C05441=1094.407,-79.945,449.901,175.167,15.277,152.247
C05442=1094.413,-79.695,449.891,175.169,15.278,152.247
C05443=1094.419,-79.446,449.880,175.170,15.279,152.247
C05444=1094.425,-79.197,449.869,175.172,15.279,152.247
C05445=1094.431,-78.946,449.859,175.174,15.280,152.246
C05446=1094.437,-78.696,449.848,175.175,15.280,152.246
C05447=1094.443,-78.447,449.837,175.177,15.281,152.246
C05448=1094.448,-78.197,449.826,175.179,15.282,152.246
C05449=1094.455,-77.947,449.815,175.181,15.283,152.246
C05450=1094.461,-77.698,449.805,175.182,15.284,152.245
C05451=1094.467,-77.449,449.794,175.183,15.284,152.245
C05452=1094.473,-77.199,449.783,175.185,15.285,152.245
C05453=1094.479,-76.948,449.772,175.187,15.286,152.245
C05454=1094.484,-76.699,449.762,175.189,15.286,152.244
C05455=1094.490,-76.449,449.751,175.191,15.287,152.244
C05456=1094.497,-76.200,449.740,175.192,15.288,152.244
C05457=1094.503,-75.950,449.729,175.194,15.288,152.244
C05458=1094.509,-75.700,449.718,175.195,15.289,152.244
C05459=1094.515,-75.451,449.707,175.197,15.290,152.243
C05460=1094.521,-75.201,449.696,175.199,15.291,152.243
C05461=1094.527,-74.951,449.685,175.201,15.291,152.243
C05462=1094.532,-74.702,449.674,175.203,15.292,152.243
C05463=1094.539,-74.453,449.664,175.204,15.292,152.242
C05464=1094.545,-74.202,449.653,175.205,15.293,152.242
C05465=1094.551,-73.953,449.642,175.207,15.294,152.242
C05466=1094.557,-73.703,449.631,175.209,15.295,152.242
C05467=1094.562,-73.453,449.621,175.211,15.296,152.242
C05468=1094.568,-73.203,449.610,175.213,15.297,152.241
C05469=1094.574,-72.954,449.599,175.214,15.297,152.241
C05470=1094.580,-72.704,449.588,175.215,15.298,152.241
C05471=1094.586,-72.455,449.577,175.217,15.299,152.241
C05472=1094.592,-72.204,449.566,175.219,15.299,152.241
C05473=1094.597,-71.955,449.554,175.221,15.301,152.241
C05474=1094.603,-71.705,449.543,175.223,15.301,152.240
C05475=1094.608,-71.456,449.533,175.224,15.302,152.240
C05476=1094.615,-71.205,449.521,175.225,15.302,152.240
C05477=1094.621,-70.956,449.510,175.227,15.303,152.240
C05478=1094.627,-70.707,449.499,175.229,15.304,152.239
C05479=1094.633,-70.457,449.488,175.231,15.305,152.239
C05480=1094.639,-70.207,449.477,175.233,15.306,152.239
C05481=1094.644,-69.958,449.466,175.234,15.306,152.239
C05482=1094.650,-69.708,449.455,175.236,15.308,152.239
C05483=1094.656,-69.458,449.444,175.237,15.308,152.238
C05484=1094.662,-69.209,449.433,175.239,15.308,152.238
C05485=1094.668,-68.959,449.422,175.241,15.310,152.238
C05486=1094.674,-68.709,449.411,175.242,15.310,152.238
C05487=1094.680,-68.460,449.400,175.244,15.311,152.238
C05488=1094.685,-68.210,449.388,175.246,15.312,152.237
C05489=1094.691,-67.960,449.377,175.248,15.313,152.237
C05490=1094.697,-67.710,449.366,175.250,15.314,152.237
C05491=1094.703,-67.461,449.355,175.250,15.314,152.237
C05492=1094.709,-67.211,449.343,175.252,15.315,152.237
C05493=1094.715,-66.962,449.333,175.254,15.316,152.236
C05494=1094.721,-66.712,449.322,175.256,15.317,152.236
C05495=1094.727,-66.462,449.310,175.258,15.317,152.236
C05496=1094.733,-66.212,449.300,175.260,15.318,152.236
C05497=1094.739,-65.963,449.289,175.261,15.319,152.236
C05498=1094.745,-65.713,449.276,175.263,15.320,152.235
C05499=1094.750,-65.464,449.265,175.264,15.321,152.235
C05500=1094.757,-65.213,449.254,175.266,15.321,152.235
C05501=1094.763,-64.943,449.242,175.268,15.322,152.235
C05502=1094.769,-64.674,449.231,175.270,15.323,152.235
C05503=1094.776,-64.404,449.218,175.272,15.324,152.234
C05504=1094.782,-64.134,449.206,175.274,15.325,152.234
C05505=1094.788,-63.884,449.194,175.275,15.325,152.234
C05506=1094.794,-63.634,449.184,175.277,15.326,152.234
C05507=1094.801,-63.385,449.172,175.278,15.327,152.234
C05508=1094.806,-63.135,449.161,175.280,15.328,152.233
C05509=1094.811,-62.885,449.149,175.282,15.329,152.233
C05510=1094.818,-62.635,449.138,175.284,15.330,152.233
C05511=1094.824,-62.386,449.126,175.286,15.330,152.233
C05512=1094.830,-62.136,449.115,175.287,15.332,152.233
C05513=1094.836,-61.887,449.104,175.289,15.332,152.232
C05514=1094.842,-61.636,449.093,175.291,15.333,152.232
C05515=1094.847,-61.387,449.081,175.292,15.334,152.232
C05516=1094.853,-61.138,449.070,175.294,15.334,152.232
C05517=1094.860,-60.888,449.059,175.295,15.335,152.232
C05518=1094.866,-60.639,449.047,175.297,15.336,152.231
C05519=1094.872,-60.389,449.036,175.299,15.337,152.231
C05520=1094.878,-60.139,449.025,175.301,15.338,152.231
C05521=1094.884,-59.889,449.012,175.303,15.339,152.231
C05522=1094.889,-59.640,449.002,175.304,15.339,152.230
C05523=1094.896,-59.390,448.990,175.306,15.341,152.230
C05524=1094.902,-59.141,448.979,175.308,15.341,152.230
C05525=1094.908,-58.890,448.968,175.310,15.342,152.230
C05526=1094.913,-58.641,448.956,175.311,15.343,152.230
C05527=1094.919,-58.392,448.944,175.312,15.343,152.229
C05528=1094.925,-58.142,448.933,175.314,15.344,152.229
C05529=1094.931,-57.892,448.922,175.316,15.345,152.229
C05530=1094.937,-57.642,448.910,175.318,15.346,152.229
C05531=1094.943,-57.393,448.899,175.320,15.346,152.229
C05532=1094.949,-57.143,448.887,175.321,15.348,152.228
C05533=1094.955,-56.894,448.876,175.323,15.348,152.228
C05534=1094.962,-56.643,448.865,175.325,15.349,152.228
C05535=1094.967,-56.394,448.853,175.327,15.350,152.228
C05536=1094.973,-56.144,448.841,175.329,15.351,152.228
C05537=1094.980,-55.895,448.829,175.330,15.352,152.227
C05538=1094.986,-55.645,448.819,175.332,15.353,152.227
C05539=1094.991,-55.395,448.806,175.334,15.354,152.227
C05540=1094.997,-55.146,448.795,175.336,15.354,152.227
C05541=1095.004,-54.896,448.783,175.337,15.355,152.227
C05542=1095.010,-54.647,448.772,175.339,15.355,152.226
C05543=1095.015,-54.397,448.760,175.340,15.356,152.226
C05544=1095.021,-54.147,448.749,175.342,15.357,152.226
C05545=1095.028,-53.898,448.737,175.344,15.358,152.226
C05546=1095.033,-53.648,448.725,175.346,15.359,152.225
C05547=1095.040,-53.398,448.713,175.347,15.360,152.225
C05548=1095.046,-53.148,448.702,175.349,15.361,152.225
C05549=1095.052,-52.899,448.691,175.351,15.361,152.225
C05550=1095.058,-52.649,448.679,175.353,15.363,152.225
C05551=1095.064,-52.400,448.667,175.355,15.363,152.224
C05552=1095.070,-52.150,448.656,175.356,15.364,152.224
C05553=1095.076,-51.901,448.644,175.358,15.365,152.224
C05554=1095.082,-51.650,448.633,175.360,15.366,152.224
C05555=1095.088,-51.401,448.621,175.362,15.367,152.224
C05556=1095.094,-51.151,448.610,175.363,15.368,152.223
C05557=1095.100,-50.901,448.597,175.365,15.368,152.223
C05558=1095.106,-50.652,448.586,175.367,15.370,152.223
C05559=1095.112,-50.402,448.574,175.369,15.370,152.223
C05560=1095.118,-50.153,448.562,175.371,15.371,152.223
C05561=1095.124,-49.903,448.551,175.371,15.372,152.223
C05562=1095.129,-49.654,448.539,175.373,15.372,152.222
C05563=1095.136,-49.404,448.527,175.375,15.373,152.222
C05564=1095.141,-49.154,448.515,175.377,15.374,152.222
C05565=1095.147,-48.885,448.503,175.379,15.376,152.222
C05566=1095.153,-48.616,448.489,175.381,15.377,152.222
C05567=1095.160,-48.347,448.477,175.383,15.377,152.221
C05568=1095.166,-48.080,448.464,175.385,15.378,152.221
C05569=1095.172,-47.829,448.452,175.386,15.379,152.221
C05570=1095.178,-47.580,448.441,175.388,15.380,152.221
C05571=1095.184,-47.330,448.428,175.390,15.381,152.221
C05572=1095.190,-47.080,448.417,175.392,15.382,152.220
C05573=1095.195,-46.831,448.405,175.393,15.383,152.220
C05574=1095.202,-46.581,448.393,175.395,15.384,152.220
C05575=1095.207,-46.332,448.381,175.397,15.385,152.220
C05576=1095.214,-46.082,448.369,175.399,15.386,152.220
C05577=1095.219,-45.833,448.357,175.400,15.387,152.219
C05578=1095.225,-45.583,448.345,175.402,15.387,152.219
C05579=1095.231,-45.333,448.333,175.404,15.388,152.219
C05580=1095.237,-45.084,448.321,175.406,15.389,152.219
C05581=1095.243,-44.834,448.309,175.408,15.390,152.219
C05582=1095.248,-44.584,448.298,175.409,15.391,152.218
C05583=1095.255,-44.335,448.286,175.411,15.392,152.218
C05584=1095.261,-44.085,448.273,175.413,15.393,152.218
C05585=1095.266,-43.836,448.261,175.415,15.394,152.218
C05586=1095.272,-43.585,448.250,175.416,15.394,152.218
C05587=1095.278,-43.335,448.237,175.418,15.396,152.217
C05588=1095.284,-43.087,448.226,175.420,15.396,152.217
C05589=1095.290,-42.837,448.213,175.421,15.398,152.217
C05590=1095.295,-42.587,448.202,175.423,15.398,152.217
C05591=1095.302,-42.337,448.190,175.425,15.399,152.217
C05592=1095.308,-42.087,448.177,175.427,15.400,152.216
C05593=1095.313,-41.838,448.165,175.429,15.401,152.216
C05594=1095.320,-41.589,448.153,175.430,15.402,152.216
C05595=1095.326,-41.339,448.140,175.432,15.403,152.216
C05596=1095.331,-41.089,448.129,175.434,15.404,152.216
C05597=1095.337,-40.839,448.117,175.436,15.405,152.216
C05598=1095.343,-40.590,448.104,175.438,15.405,152.215
C05599=1095.349,-40.341,448.093,175.439,15.406,152.215
C05600=1095.355,-40.091,448.080,175.441,15.407,152.215
C05601=1095.361,-39.841,448.068,175.443,15.408,152.215
C05602=1095.367,-39.591,448.057,175.445,15.409,152.215
C05603=1095.373,-39.342,448.044,175.446,15.410,152.214
C05604=1095.379,-39.092,448.032,175.448,15.411,152.214
C05605=1095.385,-38.842,448.020,175.450,15.412,152.214
C05606=1095.391,-38.593,448.008,175.451,15.413,152.214
C05607=1095.397,-38.343,447.995,175.453,15.414,152.214
C05608=1095.402,-38.094,447.983,175.455,15.415,152.213
C05609=1095.409,-37.844,447.971,175.457,15.415,152.213
C05610=1095.414,-37.594,447.958,175.458,15.417,152.213
C05611=1095.420,-37.345,447.946,175.460,15.417,152.213
C05612=1095.425,-37.095,447.934,175.462,15.418,152.213
C05613=1095.431,-36.845,447.922,175.464,15.419,152.212
C05614=1095.437,-36.596,447.910,175.466,15.420,152.212
C05615=1095.443,-36.346,447.898,175.467,15.421,152.212
C05616=1095.449,-36.096,447.885,175.469,15.422,152.212
C05617=1095.454,-35.847,447.873,175.471,15.424,152.212
C05618=1095.460,-35.597,447.860,175.473,15.424,152.211
C05619=1095.467,-35.348,447.848,175.475,15.425,152.211
C05620=1095.473,-35.098,447.836,175.477,15.426,152.211
C05621=1095.478,-34.848,447.824,175.478,15.427,152.211
C05622=1095.484,-34.599,447.811,175.480,15.428,152.211
C05623=1095.490,-34.349,447.798,175.482,15.429,152.211
C05624=1095.495,-34.100,447.786,175.484,15.430,152.210
C05625=1095.501,-33.850,447.774,175.486,15.431,152.210
C05626=1095.508,-33.600,447.762,175.487,15.432,152.210
C05627=1095.514,-33.350,447.749,175.489,15.433,152.210
C05628=1095.519,-33.101,447.737,175.491,15.434,152.210
C05629=1095.526,-32.832,447.724,175.493,15.434,152.209
C05630=1095.532,-32.564,447.710,175.494,15.436,152.209
C05631=1095.538,-32.296,447.696,175.497,15.437,152.209
C05632=1095.545,-32.028,447.683,175.499,15.438,152.209
C05633=1095.550,-31.769,447.670,175.500,15.439,152.209
C05634=1095.557,-31.512,447.658,175.502,15.439,152.208
C05635=1095.563,-31.253,447.645,175.504,15.441,152.208
C05636=1095.569,-30.996,447.631,175.506,15.441,152.208
C05637=1095.575,-30.746,447.619,175.507,15.443,152.208
C05638=1095.581,-30.497,447.607,175.510,15.444,152.208
C05639=1095.587,-30.247,447.594,175.512,15.445,152.207
C05640=1095.593,-29.997,447.582,175.513,15.446,152.207
C05641=1095.598,-29.747,447.569,175.515,15.446,152.207
C05642=1095.604,-29.498,447.557,175.517,15.448,152.207
C05643=1095.610,-29.249,447.544,175.519,15.448,152.207
C05644=1095.616,-28.999,447.531,175.521,15.449,152.206
C05645=1095.622,-28.749,447.519,175.522,15.450,152.206
C05646=1095.628,-28.499,447.506,175.524,15.451,152.206
C05647=1095.633,-28.250,447.494,175.526,15.452,152.206
C05648=1095.640,-28.001,447.481,175.528,15.453,152.206
C05649=1095.646,-27.751,447.469,175.529,15.454,152.206
C05650=1095.652,-27.501,447.456,175.531,15.455,152.205
C05651=1095.658,-27.251,447.444,175.533,15.455,152.205
C05652=1095.664,-27.002,447.431,175.535,15.457,152.205
C05653=1095.669,-26.753,447.418,175.537,15.458,152.205
C05654=1095.675,-26.503,447.406,175.539,15.459,152.205
C05655=1095.681,-26.253,447.393,175.541,15.460,152.204
C05656=1095.686,-26.003,447.380,175.542,15.461,152.204
C05657=1095.692,-25.754,447.367,175.544,15.462,152.204
C05658=1095.698,-25.505,447.354,175.546,15.463,152.204
C05659=1095.704,-25.255,447.342,175.548,15.464,152.204
C05660=1095.709,-25.005,447.329,175.550,15.464,152.203
C05661=1095.716,-24.756,447.316,175.551,15.465,152.203
C05662=1095.722,-24.506,447.304,175.553,15.466,152.203
C05663=1095.727,-24.256,447.291,175.555,15.468,152.203
C05664=1095.733,-24.007,447.279,175.557,15.469,152.203
C05665=1095.739,-23.757,447.266,175.559,15.470,152.202
C05666=1095.744,-23.507,447.252,175.561,15.471,152.202
C05667=1095.750,-23.257,447.240,175.562,15.472,152.202
C05668=1095.756,-23.008,447.227,175.564,15.472,152.202
C05669=1095.762,-22.759,447.214,175.566,15.474,152.202
C05670=1095.768,-22.509,447.202,175.568,15.474,152.201
C05671=1095.774,-22.260,447.189,175.570,15.475,152.201
C05672=1095.780,-22.010,447.176,175.572,15.477,152.201
C05673=1095.786,-21.760,447.163,175.574,15.477,152.201
C05674=1095.791,-21.510,447.150,175.575,15.479,152.201
C05675=1095.796,-21.261,447.137,175.577,15.479,152.200
C05676=1095.803,-21.012,447.124,175.579,15.481,152.200
C05677=1095.808,-20.762,447.112,175.581,15.481,152.200
C05678=1095.814,-20.512,447.099,175.583,15.482,152.200
C05679=1095.821,-20.263,447.086,175.584,15.483,152.200
C05680=1095.826,-20.013,447.073,175.586,15.484,152.200
C05681=1095.832,-19.763,447.059,175.588,15.486,152.199
C05682=1095.838,-19.514,447.047,175.590,15.486,152.199
C05683=1095.844,-19.264,447.034,175.592,15.488,152.199
C05684=1095.850,-19.014,447.021,175.594,15.488,152.199
C05685=1095.855,-18.765,447.009,175.596,15.489,152.199
C05686=1095.861,-18.516,446.995,175.597,15.490,152.198
C05687=1095.867,-18.266,446.982,175.599,15.491,152.198
C05688=1095.873,-18.016,446.969,175.601,15.492,152.198
C05689=1095.879,-17.767,446.957,175.603,15.493,152.198
C05690=1095.885,-17.517,446.943,175.605,15.494,152.197
C05691=1095.890,-17.267,446.930,175.607,15.495,152.197
C05692=1095.896,-17.018,446.917,175.609,15.496,152.197
C05693=1095.902,-16.757,446.903,175.610,15.497,152.197
C05694=1095.909,-16.496,446.889,175.612,15.498,152.197
C05695=1095.915,-16.235,446.876,175.614,15.499,152.197
C05696=1095.921,-15.975,446.862,175.617,15.500,152.196
C05697=1095.927,-15.725,446.850,175.618,15.501,152.196
C05698=1095.933,-15.476,446.836,175.620,15.502,152.196
C05699=1095.939,-15.226,446.824,175.622,15.503,152.196
C05700=1095.944,-14.976,446.810,175.624,15.504,152.196
C05701=1095.950,-14.726,446.797,175.625,15.505,152.195
C05702=1095.956,-14.477,446.784,175.628,15.506,152.195
C05703=1095.961,-14.227,446.771,175.630,15.507,152.195
C05704=1095.968,-13.977,446.758,175.631,15.508,152.195
C05705=1095.974,-13.728,446.744,175.633,15.509,152.195
C05706=1095.979,-13.478,446.731,175.635,15.510,152.194
C05707=1095.985,-13.229,446.718,175.637,15.511,152.194
C05708=1095.990,-12.979,446.705,175.638,15.512,152.194
C05709=1095.997,-12.729,446.692,175.641,15.513,152.194
C05710=1096.003,-12.480,446.678,175.643,15.514,152.194
C05711=1096.008,-12.230,446.665,175.645,15.515,152.193
C05712=1096.014,-11.981,446.652,175.646,15.516,152.193
C05713=1096.019,-11.732,446.638,175.648,15.517,152.193
C05714=1096.025,-11.482,446.626,175.650,15.518,152.193
C05715=1096.031,-11.233,446.613,175.652,15.519,152.193
C05716=1096.037,-10.983,446.599,175.654,15.520,152.192
C05717=1096.043,-10.733,446.586,175.656,15.521,152.192
C05718=1096.048,-10.484,446.572,175.658,15.522,152.192
C05719=1096.054,-10.234,446.559,175.660,15.523,152.192
C05720=1096.059,-9.984,446.546,175.661,15.524,152.192
C05721=1096.066,-9.735,446.533,175.663,15.525,152.191
C05722=1096.072,-9.486,446.519,175.666,15.526,152.191
C05723=1096.077,-9.236,446.505,175.667,15.527,152.191
C05724=1096.083,-8.986,446.493,175.669,15.528,152.191
C05725=1096.089,-8.737,446.479,175.671,15.528,152.191
C05726=1096.095,-8.487,446.466,175.673,15.530,152.190
C05727=1096.100,-8.238,446.452,175.675,15.530,152.190
C05728=1096.107,-7.987,446.439,175.677,15.532,152.190
C05729=1096.112,-7.738,446.425,175.679,15.533,152.190
C05730=1096.119,-7.488,446.412,175.681,15.534,152.190
C05731=1096.124,-7.239,446.398,175.682,15.535,152.189
C05732=1096.130,-6.989,446.385,175.684,15.535,152.189
C05733=1096.136,-6.739,446.372,175.686,15.536,152.189
C05734=1096.142,-6.490,446.358,175.688,15.538,152.189
C05735=1096.147,-6.240,446.344,175.690,15.539,152.189
C05736=1096.153,-5.991,446.331,175.692,15.539,152.188
C05737=1096.159,-5.742,446.317,175.694,15.541,152.188
C05738=1096.165,-5.492,446.305,175.696,15.541,152.188
C05739=1096.170,-5.242,446.291,175.698,15.542,152.188
C05740=1096.176,-4.993,446.278,175.700,15.544,152.188
C05741=1096.182,-4.743,446.264,175.702,15.544,152.187
C05742=1096.188,-4.494,446.250,175.704,15.545,152.187
C05743=1096.194,-4.244,446.236,175.705,15.546,152.187
C05744=1096.200,-3.994,446.223,175.707,15.547,152.187
C05745=1096.206,-3.745,446.209,175.709,15.548,152.186
C05746=1096.212,-3.495,446.197,175.711,15.549,152.186
C05747=1096.217,-3.245,446.183,175.713,15.550,152.186
C05748=1096.224,-2.996,446.169,175.715,15.551,152.186
C05749=1096.229,-2.747,446.156,175.717,15.552,152.186
C05750=1096.234,-2.497,446.142,175.719,15.553,152.185
C05751=1096.240,-2.247,446.128,175.721,15.555,152.185
C05752=1096.246,-1.998,446.115,175.723,15.555,152.185
C05753=1096.252,-1.749,446.101,175.725,15.556,152.185
C05754=1096.257,-1.499,446.087,175.726,15.557,152.185
C05755=1096.263,-1.250,446.074,175.728,15.558,152.184
C05756=1096.269,-1.000,446.060,175.731,15.560,152.184
C05757=1096.275,-0.729,446.045,175.732,15.560,152.184
C05758=1096.281,-0.458,446.030,175.734,15.561,152.184
C05759=1096.288,-0.188,446.015,175.737,15.563,152.184
C05760=1096.294,0.084,446.000,175.739,15.564,152.183
C05761=1096.299,0.333,445.987,175.741,15.564,152.183
C05762=1096.305,0.583,445.973,175.743,15.566,152.183
C05763=1096.312,0.833,445.959,175.745,15.567,152.183
C05764=1096.317,1.082,445.945,175.747,15.568,152.182
C05765=1096.322,1.332,445.931,175.748,15.569,152.182
C05766=1096.328,1.581,445.918,175.750,15.569,152.182
C05767=1096.333,1.831,445.904,175.753,15.571,152.182
C05768=1096.340,2.080,445.890,175.754,15.572,152.182
C05769=1096.345,2.329,445.876,175.756,15.573,152.181
C05770=1096.351,2.579,445.862,175.758,15.573,152.181
C05771=1096.357,2.829,445.848,175.760,15.574,152.181
C05772=1096.363,3.078,445.834,175.762,15.576,152.181
C05773=1096.369,3.328,445.821,175.764,15.577,152.181
C05774=1096.374,3.577,445.807,175.766,15.578,152.181
C05775=1096.380,3.827,445.793,175.768,15.578,152.180
C05776=1096.385,4.077,445.779,175.770,15.579,152.180
C05777=1096.391,4.326,445.766,175.772,15.580,152.180
C05778=1096.398,4.576,445.751,175.774,15.582,152.180
C05779=1096.403,4.825,445.737,175.776,15.582,152.179
C05780=1096.409,5.075,445.723,175.778,15.583,152.179
C05781=1096.414,5.324,445.709,175.780,15.585,152.179
C05782=1096.420,5.574,445.696,175.782,15.586,152.179
C05783=1096.426,5.824,445.682,175.784,15.586,152.178
C05784=1096.432,6.073,445.667,175.786,15.587,152.178
C05785=1096.438,6.322,445.653,175.787,15.588,152.178
C05786=1096.443,6.572,445.639,175.790,15.589,152.178
C05787=1096.449,6.821,445.626,175.792,15.590,152.178
C05788=1096.455,7.071,445.612,175.793,15.591,152.177
C05789=1096.461,7.320,445.597,175.795,15.592,152.177
C05790=1096.467,7.570,445.583,175.798,15.593,152.177
C05791=1096.472,7.820,445.570,175.800,15.594,152.177
C05792=1096.478,8.070,445.555,175.801,15.595,152.177
C05793=1096.484,8.319,445.541,175.803,15.596,152.176
C05794=1096.489,8.568,445.527,175.805,15.597,152.176
C05795=1096.496,8.818,445.514,175.808,15.598,152.176
C05796=1096.502,9.068,445.499,175.810,15.599,152.176
C05797=1096.508,9.317,445.485,175.811,15.600,152.175
C05798=1096.513,9.566,445.471,175.813,15.601,152.175
C05799=1096.519,9.816,445.457,175.816,15.602,152.175
C05800=1096.525,10.066,445.442,175.818,15.603,152.175
C05801=1096.530,10.315,445.428,175.819,15.604,152.175
C05802=1096.536,10.565,445.414,175.821,15.604,152.174
C05803=1096.542,10.814,445.400,175.824,15.606,152.174
C05804=1096.548,11.064,445.386,175.826,15.606,152.174
C05805=1096.554,11.313,445.372,175.828,15.607,152.173
C05806=1096.560,11.562,445.358,175.829,15.608,152.173
C05807=1096.566,11.813,445.344,175.832,15.610,152.173
C05808=1096.571,12.062,445.330,175.834,15.610,152.173
C05809=1096.577,12.311,445.315,175.836,15.611,152.173
C05810=1096.583,12.561,445.301,175.838,15.612,152.172
C05811=1096.589,12.810,445.286,175.840,15.613,152.172
C05812=1096.594,13.060,445.272,175.842,15.614,152.172
C05813=1096.600,13.310,445.258,175.844,15.615,152.172
C05814=1096.606,13.559,445.244,175.846,15.616,152.171
C05815=1096.612,13.809,445.230,175.848,15.616,152.171
C05816=1096.618,14.058,445.215,175.850,15.618,152.171
C05817=1096.624,14.308,445.202,175.852,15.618,152.171
C05818=1096.629,14.557,445.186,175.854,15.619,152.170
C05819=1096.635,14.807,445.172,175.856,15.620,152.170
C05820=1096.641,15.056,445.158,175.858,15.622,152.170
C05821=1096.648,15.329,445.142,175.860,15.622,152.170
C05822=1096.654,15.601,445.127,175.863,15.624,152.169
C05823=1096.660,15.874,445.111,175.865,15.624,152.169
C05824=1096.667,16.147,445.095,175.867,15.626,152.169
C05825=1096.672,16.397,445.081,175.869,15.627,152.169
C05826=1096.678,16.646,445.066,175.871,15.628,152.169
C05827=1096.684,16.896,445.052,175.873,15.628,152.168
C05828=1096.689,17.145,445.037,175.875,15.630,152.168
C05829=1096.695,17.395,445.023,175.877,15.630,152.168
C05830=1096.701,17.645,445.008,175.879,15.631,152.167
C05831=1096.706,17.894,444.994,175.881,15.632,152.167
C05832=1096.712,18.143,444.980,175.883,15.634,152.167
C05833=1096.718,18.393,444.965,175.885,15.634,152.167
C05834=1096.724,18.642,444.951,175.887,15.635,152.167
C05835=1096.730,18.891,444.936,175.890,15.636,152.166
C05836=1096.735,19.142,444.921,175.892,15.637,152.166
C05837=1096.741,19.391,444.907,175.894,15.638,152.166
C05838=1096.747,19.641,444.893,175.896,15.638,152.166
C05839=1096.753,19.890,444.878,175.898,15.640,152.165
C05840=1096.759,20.139,444.864,175.900,15.641,152.165
C05841=1096.765,20.389,444.849,175.902,15.642,152.165
C05842=1096.770,20.639,444.834,175.904,15.642,152.165
C05843=1096.776,20.888,444.820,175.906,15.644,152.164
C05844=1096.782,21.138,444.805,175.908,15.644,152.164
C05845=1096.787,21.387,444.791,175.910,15.645,152.164
C05846=1096.793,21.637,444.775,175.913,15.646,152.164
C05847=1096.799,21.886,444.761,175.914,15.648,152.163
C05848=1096.804,22.135,444.747,175.916,15.648,152.163
C05849=1096.811,22.385,444.732,175.918,15.649,152.163
C05850=1096.815,22.635,444.717,175.921,15.650,152.163
C05851=1096.822,22.885,444.702,175.923,15.651,152.162
C05852=1096.828,23.134,444.688,175.925,15.652,152.162
C05853=1096.832,23.383,444.673,175.927,15.653,152.162
C05854=1096.839,23.633,444.658,175.929,15.654,152.162
C05855=1096.844,23.882,444.644,175.931,15.654,152.161
C05856=1096.851,24.132,444.629,175.933,15.655,152.161
C05857=1096.856,24.382,444.614,175.936,15.656,152.161
C05858=1096.862,24.631,444.599,175.937,15.658,152.161
C05859=1096.868,24.880,444.585,175.939,15.658,152.161
C05860=1096.873,25.130,444.569,175.942,15.660,152.160
C05861=1096.879,25.379,444.555,175.944,15.660,152.160
C05862=1096.885,25.629,444.541,175.945,15.661,152.160
C05863=1096.890,25.879,444.525,175.947,15.662,152.159
C05864=1096.896,26.128,444.511,175.950,15.663,152.159
C05865=1096.902,26.377,444.496,175.952,15.664,152.159
C05866=1096.908,26.627,444.481,175.954,15.665,152.159
C05867=1096.914,26.876,444.466,175.956,15.666,152.158
C05868=1096.919,27.126,444.452,175.958,15.667,152.158
C05869=1096.925,27.376,444.436,175.960,15.667,152.158
C05870=1096.931,27.625,444.422,175.963,15.669,152.158
C05871=1096.937,27.874,444.407,175.965,15.669,152.157
C05872=1096.942,28.124,444.392,175.967,15.670,152.157
C05873=1096.949,28.373,444.377,175.969,15.671,152.157
C05874=1096.954,28.622,444.362,175.971,15.672,152.157
C05875=1096.960,28.872,444.347,175.973,15.673,152.156
C05876=1096.966,29.122,444.333,175.975,15.673,152.156
C05877=1096.971,29.372,444.317,175.978,15.675,152.156
C05878=1096.977,29.621,444.303,175.980,15.676,152.155
C05879=1096.983,29.871,444.287,175.981,15.676,152.155
C05880=1096.988,30.120,444.272,175.984,15.678,152.155
C05881=1096.994,30.370,444.257,175.986,15.678,152.155
C05882=1097.000,30.619,444.242,175.988,15.679,152.154
C05883=1097.005,30.868,444.227,175.991,15.680,152.154
C05884=1097.011,31.117,444.212,175.992,15.681,152.154
C05885=1097.017,31.392,444.195,175.994,15.682,152.154
C05886=1097.023,31.666,444.179,175.997,15.683,152.153
C05887=1097.030,31.940,444.162,176.000,15.684,152.153
C05888=1097.037,32.214,444.146,176.002,15.685,152.153
C05889=1097.042,32.464,444.130,176.003,15.686,152.153
C05890=1097.048,32.713,444.116,176.006,15.687,152.152
C05891=1097.054,32.963,444.100,176.008,15.688,152.152
C05892=1097.059,33.212,444.085,176.010,15.688,152.152
C05893=1097.065,33.462,444.070,176.013,15.689,152.151
C05894=1097.070,33.711,444.055,176.015,15.690,152.151
C05895=1097.076,33.961,444.040,176.017,15.691,152.151
C05896=1097.082,34.211,444.025,176.019,15.692,152.151
C05897=1097.088,34.460,444.010,176.021,15.693,152.150
C05898=1097.094,34.709,443.994,176.023,15.694,152.150
C05899=1097.100,34.958,443.979,176.026,15.695,152.150
C05900=1097.105,35.208,443.964,176.028,15.696,152.150
C05901=1097.111,35.457,443.949,176.030,15.696,152.149
C05902=1097.117,35.707,443.933,176.032,15.698,152.149
C05903=1097.122,35.957,443.918,176.034,15.698,152.149
C05904=1097.128,36.206,443.903,176.036,15.699,152.148
C05905=1097.134,36.456,443.888,176.039,15.700,152.148
C05906=1097.140,36.704,443.872,176.041,15.701,152.148
C05907=1097.145,36.954,443.857,176.043,15.701,152.148
C05908=1097.151,37.204,443.841,176.045,15.703,152.147
C05909=1097.157,37.453,443.827,176.047,15.703,152.147
C05910=1097.163,37.703,443.811,176.049,15.704,152.147
C05911=1097.169,37.952,443.796,176.052,15.705,152.146
C05912=1097.174,38.201,443.780,176.054,15.706,152.146
C05913=1097.180,38.451,443.765,176.056,15.706,152.146
C05914=1097.185,38.701,443.750,176.059,15.708,152.146
C05915=1097.191,38.950,443.735,176.060,15.708,152.145
C05916=1097.197,39.200,443.719,176.062,15.709,152.145
C05917=1097.202,39.449,443.703,176.065,15.710,152.145
C05918=1097.209,39.699,443.688,176.067,15.711,152.144
C05919=1097.214,39.948,443.673,176.069,15.712,152.144
C05920=1097.220,40.197,443.657,176.072,15.713,152.144
C05921=1097.225,40.447,443.641,176.074,15.713,152.144
C05922=1097.231,40.696,443.627,176.076,15.714,152.143
C05923=1097.237,40.945,443.611,176.078,15.715,152.143
C05924=1097.243,41.195,443.595,176.080,15.716,152.143
C05925=1097.248,41.445,443.580,176.083,15.717,152.142
C05926=1097.253,41.695,443.564,176.085,15.718,152.142
C05927=1097.260,41.943,443.549,176.087,15.718,152.142
C05928=1097.265,42.193,443.533,176.090,15.720,152.142
C05929=1097.271,42.442,443.517,176.091,15.720,152.141
C05930=1097.276,42.692,443.502,176.093,15.721,152.141
C05931=1097.283,42.941,443.487,176.096,15.722,152.141
C05932=1097.288,43.191,443.471,176.098,15.723,152.140
C05933=1097.294,43.441,443.455,176.100,15.723,152.140
C05934=1097.299,43.690,443.440,176.103,15.725,152.140
C05935=1097.305,43.939,443.424,176.105,15.725,152.140
C05936=1097.311,44.189,443.408,176.107,15.726,152.139
C05937=1097.316,44.438,443.392,176.109,15.727,152.139
C05938=1097.322,44.688,443.377,176.111,15.728,152.139
C05939=1097.327,44.937,443.362,176.114,15.729,152.138
C05940=1097.334,45.186,443.346,176.116,15.730,152.138
C05941=1097.339,45.436,443.331,176.118,15.730,152.138
C05942=1097.345,45.685,443.315,176.121,15.731,152.137
C05943=1097.350,45.935,443.299,176.123,15.732,152.137
C05944=1097.356,46.184,443.283,176.125,15.733,152.137
C05945=1097.361,46.433,443.268,176.127,15.734,152.137
C05946=1097.367,46.683,443.251,176.129,15.735,152.136
C05947=1097.373,46.933,443.236,176.132,15.736,152.136
C05948=1097.378,47.181,443.220,176.134,15.736,152.136
C05949=1097.384,47.456,443.202,176.137,15.738,152.135
C05950=1097.390,47.730,443.185,176.139,15.738,152.135
C05951=1097.397,48.005,443.168,176.141,15.739,152.135
C05952=1097.403,48.279,443.150,176.143,15.740,152.134
C05953=1097.408,48.528,443.135,176.146,15.741,152.134
C05954=1097.414,48.778,443.118,176.148,15.741,152.134
C05955=1097.420,49.028,443.103,176.151,15.743,152.133
C05956=1097.426,49.277,443.087,176.153,15.743,152.133
C05957=1097.431,49.526,443.071,176.155,15.744,152.133
C05958=1097.437,49.776,443.055,176.158,15.745,152.132
C05959=1097.442,50.025,443.039,176.159,15.746,152.132
C05960=1097.448,50.275,443.023,176.162,15.746,152.132
C05961=1097.453,50.524,443.007,176.164,15.747,152.132
C05962=1097.459,50.773,442.992,176.166,15.748,152.131
C05963=1097.465,51.023,442.976,176.169,15.749,152.131
C05964=1097.471,51.272,442.959,176.171,15.750,152.131
C05965=1097.476,51.521,442.944,176.173,15.750,152.130
C05966=1097.482,51.771,442.928,176.176,15.751,152.130
C05967=1097.488,52.020,442.912,176.178,15.752,152.130
C05968=1097.494,52.270,442.896,176.181,15.753,152.129
C05969=1097.500,52.519,442.880,176.183,15.753,152.129
C05970=1097.505,52.768,442.864,176.185,15.754,152.129
C05971=1097.511,53.018,442.848,176.188,15.755,152.128
C05972=1097.517,53.267,442.832,176.189,15.756,152.128
C05973=1097.522,53.517,442.815,176.192,15.757,152.128
C05974=1097.528,53.766,442.799,176.194,15.757,152.127
C05975=1097.533,54.016,442.784,176.196,15.758,152.127
C05976=1097.539,54.265,442.768,176.199,15.759,152.127
C05977=1097.545,54.514,442.751,176.201,15.760,152.126
C05978=1097.551,54.764,442.735,176.203,15.760,152.126
C05979=1097.556,55.014,442.720,176.206,15.761,152.126
C05980=1097.562,55.263,442.703,176.208,15.762,152.125
C05981=1097.568,55.512,442.687,176.211,15.763,152.125
C05982=1097.573,55.761,442.671,176.213,15.763,152.125
C05983=1097.579,56.011,442.654,176.215,15.764,152.124
C05984=1097.584,56.261,442.639,176.218,15.765,152.124
C05985=1097.590,56.510,442.623,176.220,15.765,152.124
C05986=1097.596,56.759,442.606,176.222,15.767,152.123
C05987=1097.602,57.009,442.590,176.225,15.767,152.123
C05988=1097.608,57.258,442.574,176.226,15.768,152.123
C05989=1097.614,57.507,442.558,176.229,15.768,152.122
C05990=1097.619,57.756,442.541,176.231,15.769,152.122
C05991=1097.624,58.006,442.526,176.234,15.770,152.122
C05992=1097.630,58.256,442.509,176.236,15.771,152.121
C05993=1097.636,58.505,442.493,176.238,15.771,152.121
C05994=1097.642,58.754,442.477,176.241,15.772,152.121
C05995=1097.648,59.004,442.461,176.243,15.772,152.120
C05996=1097.653,59.253,442.444,176.246,15.774,152.120
C05997=1097.659,59.503,442.427,176.248,15.774,152.120
C05998=1097.665,59.752,442.411,176.251,15.775,152.119
C05999=1097.671,60.001,442.395,176.253,15.776,152.119
C06000=1097.677,60.251,442.379,176.255,15.776,152.118
C06001=1097.683,60.500,442.362,176.258,15.777,152.118
C06002=1097.688,60.750,442.346,176.260,15.777,152.118
C06003=1097.694,60.999,442.329,176.263,15.779,152.117
C06004=1097.700,61.249,442.313,176.265,15.779,152.117
C06005=1097.706,61.498,442.297,176.267,15.779,152.117
C06006=1097.711,61.748,442.280,176.270,15.781,152.116
C06007=1097.717,61.997,442.264,176.272,15.781,152.116
C06008=1097.723,62.246,442.247,176.275,15.782,152.116
C06009=1097.729,62.496,442.231,176.277,15.782,152.115
C06010=1097.735,62.745,442.215,176.279,15.783,152.115
C06011=1097.740,62.995,442.198,176.282,15.783,152.114
C06012=1097.746,63.244,442.182,176.284,15.784,152.114
C06013=1097.753,63.517,442.164,176.287,15.785,152.114
C06014=1097.759,63.792,442.146,176.290,15.786,152.113
C06015=1097.765,64.066,442.127,176.292,15.786,152.113
C06016=1097.772,64.340,442.109,176.295,15.787,152.112
C06017=1097.777,64.590,442.093,176.297,15.788,152.112
C06018=1097.783,64.839,442.076,176.300,15.789,152.112
C06019=1097.789,65.088,442.060,176.302,15.789,152.111
C06020=1097.794,65.338,442.043,176.305,15.790,152.111
C06021=1097.801,65.587,442.026,176.307,15.790,152.111
C06022=1097.806,65.836,442.009,176.309,15.791,152.110
C06023=1097.812,66.086,441.993,176.312,15.792,152.110
C06024=1097.818,66.335,441.977,176.314,15.792,152.110
C06025=1097.823,66.585,441.960,176.317,15.793,152.109
C06026=1097.829,66.834,441.944,176.319,15.794,152.109
C06027=1097.835,67.083,441.926,176.322,15.795,152.108
C06028=1097.840,67.332,441.910,176.324,15.795,152.108
C06029=1097.846,67.582,441.893,176.326,15.796,152.108
C06030=1097.852,67.831,441.877,176.329,15.797,152.107
C06031=1097.857,68.081,441.860,176.331,15.797,152.107
C06032=1097.863,68.330,441.843,176.334,15.798,152.107
C06033=1097.868,68.579,441.826,176.336,15.798,152.106
C06034=1097.874,68.829,441.810,176.339,15.799,152.106
C06035=1097.880,69.078,441.794,176.341,15.799,152.105
C06036=1097.886,69.327,441.776,176.344,15.801,152.105
C06037=1097.892,69.576,441.760,176.346,15.801,152.105
C06038=1097.897,69.826,441.743,176.348,15.801,152.104
C06039=1097.902,70.075,441.725,176.351,15.802,152.104
C06040=1097.908,70.325,441.709,176.353,15.803,152.104
C06041=1097.914,70.574,441.692,176.356,15.804,152.103
C06042=1097.920,70.823,441.675,176.358,15.804,152.103
C06043=1097.925,71.073,441.658,176.361,15.805,152.102
C06044=1097.931,71.322,441.642,176.363,15.806,152.102
C06045=1097.937,71.571,441.625,176.366,15.806,152.102
C06046=1097.942,71.821,441.607,176.368,15.807,152.101
C06047=1097.948,72.071,441.591,176.370,15.807,152.101
C06048=1097.954,72.320,441.574,176.373,15.808,152.101
C06049=1097.960,72.569,441.557,176.375,15.808,152.100
C06050=1097.965,72.819,441.541,176.378,15.809,152.100
C06051=1097.970,73.068,441.523,176.380,15.810,152.099
C06052=1097.976,73.317,441.507,176.383,15.810,152.099
C06053=1097.982,73.566,441.489,176.385,15.811,152.099
C06054=1097.987,73.816,441.472,176.388,15.812,152.098
C06055=1097.993,74.065,441.455,176.390,15.812,152.098
C06056=1097.999,74.315,441.438,176.393,15.813,152.097
C06057=1098.004,74.565,441.421,176.395,15.813,152.097
C06058=1098.011,74.813,441.404,176.397,15.814,152.097
C06059=1098.016,75.063,441.387,176.400,15.815,152.096
C06060=1098.021,75.312,441.370,176.402,15.815,152.096
C06061=1098.027,75.561,441.354,176.405,15.816,152.095
C06062=1098.033,75.810,441.336,176.408,15.816,152.095
C06063=1098.038,76.060,441.319,176.410,15.817,152.095
C06064=1098.045,76.309,441.302,176.413,15.817,152.094
C06065=1098.050,76.559,441.285,176.416,15.818,152.094
C06066=1098.056,76.808,441.267,176.418,15.819,152.093
C06067=1098.062,77.057,441.250,176.421,15.819,152.093
C06068=1098.067,77.307,441.234,176.423,15.820,152.093
C06069=1098.073,77.556,441.216,176.425,15.820,152.092
C06070=1098.079,77.806,441.199,176.428,15.821,152.092
C06071=1098.085,78.055,441.182,176.430,15.821,152.091
C06072=1098.090,78.304,441.165,176.433,15.822,152.091
C06073=1098.096,78.553,441.147,176.435,15.823,152.091
C06074=1098.101,78.802,441.130,176.438,15.824,152.090
C06075=1098.108,79.052,441.113,176.440,15.824,152.090
C06076=1098.113,79.302,441.096,176.443,15.825,152.089
C06077=1098.119,79.575,441.077,176.445,15.825,152.089
C06078=1098.125,79.849,441.058,176.448,15.826,152.088
C06079=1098.131,80.123,441.038,176.452,15.826,152.088
C06080=1098.137,80.397,441.020,176.455,15.827,152.087
C06081=1098.143,80.646,441.003,176.457,15.827,152.087
C06082=1098.149,80.896,440.985,176.460,15.828,152.087
C06083=1098.154,81.146,440.968,176.462,15.828,152.086
C06084=1098.160,81.395,440.950,176.465,15.829,152.086
C06085=1098.165,81.644,440.933,176.467,15.830,152.085
C06086=1098.170,81.893,440.916,176.469,15.830,152.085
C06087=1098.177,82.143,440.898,176.472,15.831,152.085
C06088=1098.183,82.392,440.881,176.475,15.831,152.084
C06089=1098.188,82.641,440.863,176.478,15.832,152.084
C06090=1098.193,82.891,440.846,176.480,15.832,152.083
C06091=1098.200,83.140,440.829,176.483,15.833,152.083
C06092=1098.205,83.389,440.811,176.485,15.833,152.082
C06093=1098.211,83.638,440.793,176.488,15.834,152.082
C06094=1098.216,83.888,440.777,176.490,15.834,152.082
C06095=1098.222,84.138,440.759,176.493,15.835,152.081
C06096=1098.227,84.387,440.741,176.495,15.835,152.081
C06097=1098.233,84.636,440.723,176.498,15.836,152.080
C06098=1098.239,84.885,440.706,176.500,15.837,152.080
C06099=1098.245,85.135,440.688,176.503,15.837,152.079
C06100=1098.250,85.384,440.671,176.505,15.838,152.079
C06101=1098.255,85.633,440.654,176.509,15.838,152.078
C06102=1098.261,85.883,440.636,176.511,15.838,152.078
C06103=1098.268,86.132,440.619,176.514,15.839,152.078
C06104=1098.273,86.381,440.601,176.516,15.839,152.077
C06105=1098.279,86.630,440.584,176.519,15.840,152.077
C06106=1098.285,86.880,440.566,176.521,15.841,152.076
C06107=1098.290,87.129,440.548,176.524,15.841,152.076
C06108=1098.296,87.378,440.530,176.527,15.841,152.075
C06109=1098.302,87.628,440.513,176.530,15.842,152.075
C06110=1098.307,87.877,440.496,176.532,15.842,152.075
C06111=1098.313,88.126,440.478,176.535,15.843,152.074
C06112=1098.319,88.376,440.460,176.537,15.843,152.074
C06113=1098.324,88.625,440.443,176.540,15.844,152.073
C06114=1098.331,88.875,440.425,176.542,15.844,152.073
C06115=1098.336,89.124,440.407,176.545,15.845,152.072
C06116=1098.341,89.373,440.389,176.548,15.845,152.072
C06117=1098.347,89.623,440.371,176.551,15.846,152.071
C06118=1098.352,89.872,440.353,176.553,15.846,152.071
C06119=1098.358,90.121,440.336,176.556,15.847,152.070
C06120=1098.364,90.371,440.318,176.558,15.847,152.070
C06121=1098.370,90.620,440.300,176.561,15.847,152.069
C06122=1098.376,90.869,440.282,176.564,15.848,152.069
C06123=1098.382,91.118,440.264,176.567,15.849,152.069
C06124=1098.387,91.367,440.247,176.569,15.849,152.068
C06125=1098.393,91.617,440.229,176.572,15.849,152.068
C06126=1098.398,91.866,440.210,176.574,15.850,152.067
C06127=1098.404,92.115,440.193,176.577,15.850,152.067
C06128=1098.410,92.365,440.175,176.579,15.851,152.066
C06129=1098.415,92.614,440.157,176.583,15.851,152.066
C06130=1098.421,92.863,440.140,176.585,15.851,152.065
C06131=1098.426,93.113,440.121,176.588,15.852,152.065
C06132=1098.432,93.362,440.104,176.590,15.852,152.065
C06133=1098.438,93.611,440.085,176.593,15.853,152.064
C06134=1098.444,93.860,440.068,176.595,15.853,152.064
C06135=1098.448,94.109,440.049,176.598,15.854,152.063
C06136=1098.454,94.359,440.031,176.601,15.854,152.063
C06137=1098.460,94.608,440.014,176.604,15.855,152.062
C06138=1098.466,94.857,439.995,176.606,15.855,152.062
C06139=1098.471,95.107,439.977,176.609,15.855,152.061
C06140=1098.477,95.356,439.960,176.612,15.856,152.061
C06141=1098.483,95.630,439.940,176.615,15.856,152.060
C06142=1098.489,95.904,439.920,176.618,15.857,152.060
C06143=1098.496,96.177,439.900,176.621,15.857,152.059
C06144=1098.502,96.451,439.880,176.623,15.858,152.059
C06145=1098.508,96.701,439.862,176.627,15.858,152.058
C06146=1098.513,96.950,439.844,176.629,15.858,152.058
C06147=1098.519,97.200,439.825,176.632,15.859,152.057
C06148=1098.524,97.449,439.808,176.634,15.859,152.057
C06149=1098.530,97.698,439.790,176.637,15.859,152.056
C06150=1098.536,97.948,439.772,176.640,15.860,152.056
C06151=1098.542,98.197,439.753,176.643,15.860,152.055
C06152=1098.547,98.446,439.735,176.645,15.860,152.055
C06153=1098.553,98.696,439.717,176.648,15.861,152.054
C06154=1098.558,98.944,439.698,176.651,15.861,152.054
C06155=1098.565,99.194,439.681,176.653,15.862,152.053
C06156=1098.570,99.443,439.662,176.656,15.862,152.053
C06157=1098.576,99.693,439.644,176.659,15.863,152.052
C06158=1098.581,99.942,439.626,176.662,15.863,152.052
C06159=1098.588,100.191,439.608,176.664,15.863,152.051
C06160=1098.592,100.440,439.589,176.668,15.864,152.051
C06161=1098.599,100.689,439.571,176.670,15.864,152.050
C06162=1098.604,100.938,439.553,176.673,15.864,152.050
C06163=1098.610,101.188,439.535,176.676,15.864,152.049
C06164=1098.616,101.438,439.516,176.679,15.865,152.049
C06165=1098.621,101.687,439.498,176.681,15.865,152.048
C06166=1098.627,101.936,439.479,176.684,15.866,152.048
C06167=1098.632,102.185,439.461,176.686,15.865,152.047
C06168=1098.639,102.434,439.442,176.689,15.866,152.047
C06169=1098.643,102.684,439.424,176.692,15.866,152.046
C06170=1098.650,102.933,439.406,176.695,15.867,152.046
C06171=1098.655,103.182,439.387,176.697,15.867,152.045
C06172=1098.661,103.431,439.369,176.700,15.868,152.045
C06173=1098.666,103.681,439.351,176.703,15.868,152.044
C06174=1098.672,103.930,439.332,176.706,15.868,152.044
C06175=1098.677,104.179,439.314,176.709,15.869,152.043
C06176=1098.683,104.428,439.295,176.711,15.869,152.043
C06177=1098.689,104.677,439.276,176.715,15.869,152.042
C06178=1098.694,104.927,439.258,176.717,15.869,152.042
C06179=1098.700,105.176,439.239,176.720,15.870,152.041
C06180=1098.705,105.426,439.221,176.722,15.870,152.041
C06181=1098.712,105.675,439.202,176.725,15.871,152.040
C06182=1098.717,105.923,439.183,176.728,15.871,152.040
C06183=1098.723,106.173,439.165,176.731,15.871,152.039
C06184=1098.728,106.422,439.147,176.733,15.871,152.039
C06185=1098.733,106.672,439.128,176.737,15.872,152.038
C06186=1098.740,106.921,439.109,176.740,15.872,152.038
C06187=1098.745,107.170,439.090,176.742,15.872,152.037
C06188=1098.751,107.420,439.073,176.745,15.873,152.037
C06189=1098.757,107.669,439.053,176.748,15.873,152.036
C06190=1098.762,107.918,439.034,176.751,15.874,152.036
C06191=1098.768,108.167,439.016,176.753,15.873,152.035
C06192=1098.773,108.416,438.998,176.757,15.874,152.034
C06193=1098.779,108.665,438.979,176.759,15.874,152.034
C06194=1098.785,108.915,438.960,176.762,15.875,152.033
C06195=1098.790,109.164,438.942,176.764,15.874,152.033
C06196=1098.796,109.413,438.923,176.768,15.875,152.032
C06197=1098.802,109.663,438.904,176.771,15.875,152.032
C06198=1098.808,109.911,438.885,176.773,15.875,152.031
C06199=1098.813,110.161,438.866,176.776,15.876,152.031
C06200=1098.819,110.411,438.848,176.779,15.876,152.030
C06201=1098.825,110.659,438.829,176.782,15.876,152.030
C06202=1098.830,110.908,438.810,176.785,15.876,152.029
C06203=1098.836,111.158,438.791,176.788,15.877,152.029
C06204=1098.842,111.407,438.772,176.790,15.877,152.028
C06205=1098.848,111.681,438.752,176.793,15.877,152.027
C06206=1098.854,111.955,438.731,176.797,15.877,152.027
C06207=1098.861,112.229,438.710,176.800,15.878,152.026
C06208=1098.867,112.503,438.690,176.804,15.878,152.025
C06209=1098.873,112.752,438.670,176.806,15.878,152.025
C06210=1098.878,113.001,438.651,176.809,15.879,152.024
C06211=1098.883,113.251,438.633,176.811,15.878,152.024
C06212=1098.889,113.501,438.614,176.815,15.879,152.023
C06213=1098.895,113.750,438.595,176.817,15.879,152.023
C06214=1098.900,113.998,438.576,176.820,15.879,152.022
C06215=1098.906,114.248,438.557,176.824,15.879,152.022
C06216=1098.912,114.497,438.538,176.826,15.880,152.021
C06217=1098.917,114.746,438.519,176.829,15.880,152.021
C06218=1098.922,114.995,438.500,176.832,15.880,152.020
C06219=1098.929,115.245,438.481,176.835,15.880,152.019
C06220=1098.935,115.494,438.462,176.837,15.880,152.019
C06221=1098.940,115.743,438.443,176.841,15.881,152.018
C06222=1098.945,115.992,438.424,176.843,15.881,152.018
C06223=1098.951,116.242,438.404,176.846,15.881,152.017
C06224=1098.956,116.490,438.385,176.849,15.882,152.017
C06225=1098.962,116.740,438.366,176.852,15.882,152.016
C06226=1098.967,116.989,438.347,176.855,15.882,152.016
C06227=1098.973,117.239,438.328,176.858,15.882,152.015
C06228=1098.978,117.487,438.309,176.861,15.882,152.014
C06229=1098.984,117.737,438.290,176.864,15.883,152.014
C06230=1098.990,117.986,438.270,176.866,15.883,152.013
C06231=1098.995,118.235,438.251,176.870,15.883,152.013
C06232=1099.000,118.484,438.232,176.872,15.883,152.012
C06233=1099.006,118.733,438.212,176.875,15.884,152.012
C06234=1099.012,118.983,438.193,176.878,15.883,152.011
C06235=1099.018,119.232,438.174,176.881,15.884,152.011
C06236=1099.023,119.481,438.155,176.884,15.884,152.010
C06237=1099.029,119.730,438.136,176.887,15.884,152.009
C06238=1099.034,119.980,438.116,176.890,15.885,152.009
C06239=1099.040,120.229,438.097,176.893,15.884,152.008
C06240=1099.046,120.478,438.077,176.896,15.885,152.008
C06241=1099.051,120.727,438.058,176.898,15.885,152.007
C06242=1099.057,120.976,438.039,176.902,15.885,152.007
C06243=1099.062,121.225,438.020,176.905,15.886,152.006
C06244=1099.068,121.475,438.001,176.907,15.885,152.005
C06245=1099.074,121.724,437.981,176.911,15.886,152.005
C06246=1099.079,121.972,437.962,176.913,15.886,152.004
C06247=1099.085,122.222,437.943,176.917,15.886,152.004
C06248=1099.091,122.471,437.923,176.920,15.886,152.003
C06249=1099.097,122.720,437.903,176.922,15.886,152.002
C06250=1099.102,122.970,437.884,176.926,15.886,152.002
C06251=1099.107,123.219,437.864,176.928,15.886,152.001
C06252=1099.113,123.468,437.844,176.931,15.887,152.001
C06253=1099.118,123.717,437.825,176.934,15.886,152.000
C06254=1099.124,123.966,437.806,176.937,15.887,152.000
C06255=1099.130,124.215,437.786,176.940,15.887,151.999
C06256=1099.136,124.465,437.767,176.943,15.887,151.998
C06257=1099.141,124.714,437.748,176.946,15.887,151.998
C06258=1099.147,124.963,437.728,176.949,15.887,151.997
C06259=1099.153,125.212,437.709,176.952,15.887,151.997
C06260=1099.159,125.462,437.689,176.956,15.888,151.996
C06261=1099.164,125.711,437.669,176.958,15.887,151.995
C06262=1099.170,125.960,437.649,176.962,15.888,151.995
C06263=1099.175,126.208,437.630,176.964,15.887,151.994
C06264=1099.181,126.458,437.611,176.967,15.888,151.994
C06265=1099.186,126.707,437.591,176.970,15.888,151.993
C06266=1099.192,126.956,437.571,176.973,15.888,151.992
C06267=1099.198,127.205,437.552,176.977,15.888,151.992
C06268=1099.204,127.454,437.532,176.979,15.888,151.991
C06269=1099.210,127.729,437.511,176.983,15.888,151.990
C06270=1099.217,128.003,437.488,176.986,15.888,151.990
C06271=1099.222,128.277,437.467,176.989,15.888,151.989
C06272=1099.229,128.550,437.446,176.993,15.888,151.988
C06273=1099.234,128.800,437.426,176.996,15.888,151.988
C06274=1099.240,129.049,437.406,176.999,15.889,151.987
C06275=1099.246,129.298,437.387,177.002,15.888,151.986
C06276=1099.252,129.547,437.367,177.005,15.888,151.986
C06277=1099.258,129.797,437.347,177.008,15.889,151.985
C06278=1099.263,130.046,437.327,177.011,15.888,151.985
C06279=1099.269,130.294,437.307,177.014,15.889,151.984
C06280=1099.274,130.544,437.288,177.017,15.888,151.983
C06281=1099.280,130.793,437.268,177.020,15.888,151.983
C06282=1099.286,131.042,437.248,177.023,15.889,151.982
C06283=1099.291,131.291,437.228,177.026,15.888,151.981
C06284=1099.297,131.540,437.208,177.030,15.889,151.981
C06285=1099.303,131.790,437.189,177.032,15.888,151.980
C06286=1099.309,132.038,437.169,177.036,15.889,151.979
C06287=1099.314,132.287,437.148,177.039,15.889,151.979
C06288=1099.320,132.537,437.129,177.042,15.888,151.978
C06289=1099.326,132.786,437.109,177.045,15.889,151.978
C06290=1099.331,133.035,437.088,177.048,15.888,151.977
C06291=1099.337,133.284,437.069,177.051,15.889,151.976
C06292=1099.342,133.533,437.049,177.054,15.889,151.976
C06293=1099.348,133.782,437.029,177.057,15.888,151.975
C06294=1099.355,134.032,437.008,177.060,15.889,151.974
C06295=1099.360,134.281,436.988,177.063,15.888,151.974
C06296=1099.366,134.530,436.968,177.066,15.889,151.973
C06297=1099.371,134.779,436.948,177.070,15.889,151.973
C06298=1099.377,135.028,436.928,177.072,15.889,151.972
C06299=1099.382,135.278,436.908,177.076,15.889,151.971
C06300=1099.388,135.527,436.888,177.079,15.889,151.970
C06301=1099.394,135.776,436.868,177.082,15.889,151.970
C06302=1099.399,136.025,436.848,177.085,15.889,151.969
C06303=1099.405,136.273,436.828,177.088,15.889,151.969
C06304=1099.410,136.523,436.808,177.091,15.889,151.968
C06305=1099.416,136.772,436.788,177.094,15.889,151.967
C06306=1099.421,137.021,436.767,177.097,15.889,151.967
C06307=1099.427,137.270,436.747,177.101,15.889,151.966
C06308=1099.433,137.520,436.726,177.103,15.888,151.965
C06309=1099.439,137.769,436.707,177.107,15.889,151.965
C06310=1099.445,138.018,436.686,177.110,15.889,151.964
C06311=1099.450,138.267,436.667,177.113,15.888,151.963
C06312=1099.455,138.516,436.646,177.116,15.889,151.963
C06313=1099.461,138.765,436.626,177.120,15.889,151.962
C06314=1099.467,139.014,436.606,177.122,15.888,151.961
C06315=1099.473,139.263,436.586,177.126,15.888,151.961
C06316=1099.479,139.513,436.565,177.128,15.888,151.960
C06317=1099.485,139.762,436.545,177.132,15.888,151.959
C06318=1099.490,140.011,436.524,177.135,15.888,151.959
C06319=1099.495,140.260,436.504,177.138,15.888,151.958
C06320=1099.501,140.509,436.484,177.141,15.888,151.957
C06321=1099.506,140.758,436.463,177.145,15.889,151.957
C06322=1099.512,141.007,436.443,177.147,15.888,151.956
C06323=1099.518,141.257,436.422,177.151,15.888,151.955
C06324=1099.523,141.506,436.402,177.154,15.888,151.955
C06325=1099.529,141.754,436.382,177.157,15.888,151.954
C06326=1099.535,142.004,436.361,177.160,15.888,151.953
C06327=1099.540,142.253,436.341,177.163,15.888,151.953
C06328=1099.546,142.502,436.321,177.167,15.888,151.952
C06329=1099.551,142.751,436.300,177.170,15.888,151.951
C06330=1099.557,143.000,436.279,177.173,15.888,151.951
C06331=1099.563,143.249,436.259,177.176,15.888,151.950
C06332=1099.569,143.498,436.238,177.180,15.888,151.949
C06333=1099.574,143.772,436.215,177.182,15.887,151.949
C06334=1099.581,144.046,436.193,177.186,15.887,151.948
C06335=1099.587,144.320,436.171,177.190,15.887,151.947
C06336=1099.593,144.594,436.147,177.193,15.887,151.946
C06337=1099.599,144.842,436.127,177.197,15.887,151.946
C06338=1099.604,145.092,436.107,177.199,15.887,151.945
C06339=1099.610,145.341,436.086,177.203,15.887,151.944
C06340=1099.616,145.590,436.066,177.207,15.887,151.943
C06341=1099.622,145.839,436.044,177.209,15.887,151.943
C06342=1099.627,146.088,436.024,177.213,15.887,151.942
C06343=1099.632,146.337,436.003,177.216,15.887,151.941
C06344=1099.639,146.586,435.983,177.219,15.886,151.941
C06345=1099.644,146.836,435.962,177.222,15.886,151.940
C06346=1099.650,147.084,435.941,177.226,15.887,151.939
C06347=1099.655,147.333,435.921,177.229,15.886,151.939
C06348=1099.662,147.583,435.900,177.232,15.886,151.938
C06349=1099.667,147.831,435.879,177.235,15.885,151.937
C06350=1099.672,148.080,435.858,177.238,15.885,151.937
C06351=1099.678,148.330,435.838,177.242,15.885,151.936
C06352=1099.684,148.579,435.816,177.244,15.885,151.935
C06353=1099.689,148.828,435.796,177.248,15.885,151.934
C06354=1099.695,149.077,435.776,177.252,15.885,151.934
C06355=1099.701,149.326,435.754,177.254,15.885,151.933
C06356=1099.706,149.575,435.734,177.258,15.885,151.932
C06357=1099.712,149.824,435.713,177.261,15.885,151.932
C06358=1099.718,150.073,435.691,177.264,15.884,151.931
C06359=1099.723,150.322,435.671,177.268,15.885,151.930
C06360=1099.729,150.571,435.650,177.271,15.885,151.930
C06361=1099.735,150.821,435.629,177.274,15.884,151.929
C06362=1099.740,151.070,435.608,177.277,15.884,151.928
C06363=1099.745,151.318,435.587,177.281,15.884,151.927
C06364=1099.751,151.567,435.566,177.284,15.883,151.927
C06365=1099.757,151.817,435.545,177.287,15.883,151.926
C06366=1099.763,152.066,435.525,177.291,15.883,151.925
C06367=1099.768,152.314,435.503,177.294,15.883,151.924
C06368=1099.774,152.564,435.482,177.297,15.883,151.924
C06369=1099.780,152.812,435.461,177.301,15.883,151.923
C06370=1099.786,153.062,435.440,177.304,15.882,151.922
C06371=1099.791,153.311,435.419,177.307,15.883,151.922
C06372=1099.796,153.560,435.398,177.310,15.882,151.921
C06373=1099.803,153.809,435.377,177.313,15.882,151.920
C06374=1099.808,154.058,435.356,177.317,15.882,151.920
C06375=1099.813,154.307,435.335,177.320,15.882,151.919
C06376=1099.819,154.556,435.314,177.323,15.882,151.918
C06377=1099.825,154.805,435.293,177.327,15.882,151.917
C06378=1099.831,155.054,435.271,177.330,15.881,151.916
C06379=1099.836,155.303,435.251,177.333,15.881,151.916
C06380=1099.841,155.552,435.229,177.337,15.881,151.915
C06381=1099.847,155.801,435.207,177.340,15.880,151.914
C06382=1099.852,156.050,435.187,177.343,15.880,151.914
C06383=1099.859,156.300,435.165,177.347,15.880,151.913
C06384=1099.864,156.549,435.144,177.350,15.880,151.912
C06385=1099.869,156.797,435.123,177.353,15.880,151.911
C06386=1099.876,157.046,435.101,177.357,15.880,151.911
C06387=1099.881,157.295,435.080,177.359,15.879,151.910
C06388=1099.887,157.545,435.059,177.363,15.879,151.909
C06389=1099.892,157.794,435.037,177.367,15.879,151.908
C06390=1099.897,158.042,435.016,177.369,15.878,151.908
C06391=1099.903,158.292,434.995,177.373,15.878,151.907
C06392=1099.909,158.540,434.974,177.376,15.879,151.906
C06393=1099.915,158.790,434.952,177.379,15.878,151.906
C06394=1099.921,159.038,434.931,177.383,15.877,151.905
C06395=1099.926,159.288,434.910,177.387,15.878,151.904
C06396=1099.931,159.537,434.888,177.390,15.878,151.903
C06397=1099.938,159.810,434.865,177.393,15.877,151.902
C06398=1099.944,160.084,434.842,177.397,15.877,151.902
C06399=1099.951,160.358,434.818,177.401,15.876,151.901
C06400=1099.957,160.631,434.793,177.404,15.876,151.900
C06401=1099.962,160.880,434.773,177.408,15.876,151.899
C06402=1099.968,161.129,434.751,177.412,15.876,151.898
C06403=1099.974,161.378,434.730,177.414,15.875,151.898
C06404=1099.979,161.628,434.708,177.418,15.875,151.897
C06405=1099.985,161.876,434.687,177.422,15.875,151.896
C06406=1099.991,162.125,434.665,177.424,15.875,151.895
C06407=1099.996,162.374,434.643,177.428,15.875,151.895
C06408=1100.001,162.623,434.622,177.432,15.874,151.894
C06409=1100.006,162.873,434.600,177.435,15.874,151.893
C06410=1100.012,163.121,434.579,177.438,15.874,151.892
C06411=1100.017,163.371,434.557,177.442,15.874,151.892
C06412=1100.023,163.619,434.535,177.445,15.874,151.891
C06413=1100.029,163.868,434.514,177.448,15.873,151.890
C06414=1100.034,164.117,434.492,177.452,15.873,151.889
C06415=1100.040,164.366,434.470,177.455,15.873,151.889
C06416=1100.045,164.615,434.448,177.458,15.872,151.888
C06417=1100.051,164.864,434.427,177.462,15.872,151.887
C06418=1100.056,165.113,434.405,177.465,15.872,151.886
C06419=1100.062,165.362,434.383,177.468,15.872,151.886
C06420=1100.067,165.611,434.361,177.472,15.871,151.885
C06421=1100.073,165.860,434.340,177.476,15.871,151.884
C06422=1100.078,166.109,434.318,177.479,15.871,151.883
C06423=1100.084,166.359,434.296,177.482,15.871,151.883
C06424=1100.089,166.607,434.274,177.486,15.870,151.882
C06425=1100.095,166.856,434.252,177.489,15.871,151.881
C06426=1100.100,167.105,434.230,177.492,15.870,151.880
C06427=1100.106,167.354,434.209,177.496,15.870,151.880
C06428=1100.112,167.603,434.186,177.500,15.870,151.879
C06429=1100.117,167.852,434.165,177.502,15.869,151.878
C06430=1100.123,168.101,434.143,177.506,15.869,151.877
C06431=1100.128,168.350,434.122,177.510,15.869,151.876
C06432=1100.134,168.599,434.099,177.513,15.869,151.876
C06433=1100.140,168.847,434.077,177.516,15.868,151.875
C06434=1100.145,169.097,434.055,177.520,15.868,151.874
C06435=1100.151,169.346,434.034,177.523,15.868,151.873
C06436=1100.156,169.595,434.012,177.526,15.867,151.873
C06437=1100.163,169.843,433.989,177.530,15.867,151.872
C06438=1100.167,170.092,433.967,177.534,15.867,151.871
C06439=1100.173,170.342,433.945,177.537,15.866,151.870
C06440=1100.179,170.591,433.924,177.540,15.866,151.869
C06441=1100.184,170.839,433.901,177.544,15.866,151.869
C06442=1100.190,171.088,433.879,177.548,15.866,151.868
C06443=1100.196,171.338,433.857,177.550,15.865,151.867
C06444=1100.202,171.586,433.835,177.554,15.865,151.866
C06445=1100.207,171.835,433.813,177.558,15.865,151.865
C06446=1100.212,172.085,433.791,177.561,15.864,151.865
C06447=1100.218,172.333,433.769,177.565,15.864,151.864
C06448=1100.224,172.582,433.746,177.568,15.863,151.863
C06449=1100.230,172.831,433.725,177.572,15.863,151.862
C06450=1100.235,173.080,433.702,177.575,15.863,151.861
C06451=1100.240,173.329,433.680,177.579,15.862,151.861
C06452=1100.247,173.578,433.658,177.582,15.862,151.860
C06453=1100.252,173.827,433.635,177.585,15.861,151.859
C06454=1100.257,174.076,433.614,177.589,15.861,151.858
C06455=1100.264,174.325,433.591,177.593,15.861,151.857
C06456=1100.269,174.574,433.569,177.597,15.861,151.856
C06457=1100.274,174.822,433.546,177.599,15.860,151.856
C06458=1100.280,175.072,433.525,177.603,15.860,151.855
C06459=1100.286,175.321,433.503,177.607,15.860,151.854
C06460=1100.291,175.570,433.480,177.610,15.859,151.853
C06461=1100.298,175.843,433.455,177.614,15.858,151.852
C06462=1100.304,176.116,433.431,177.618,15.858,151.851
C06463=1100.310,176.389,433.407,177.621,15.858,151.851
C06464=1100.316,176.662,433.382,177.625,15.857,151.850
C06465=1100.322,176.911,433.360,177.629,15.857,151.849
C06466=1100.328,177.161,433.337,177.633,15.857,151.848
C06467=1100.334,177.409,433.314,177.636,15.856,151.847
C06468=1100.340,177.659,433.293,177.640,15.855,151.846
C06469=1100.345,177.907,433.270,177.643,15.856,151.846
C06470=1100.350,178.156,433.248,177.647,15.855,151.845
C06471=1100.356,178.405,433.225,177.650,15.854,151.844
C06472=1100.362,178.654,433.203,177.654,15.854,151.843
C06473=1100.368,178.903,433.180,177.658,15.854,151.842
C06474=1100.374,179.152,433.157,177.661,15.853,151.841
C06475=1100.379,179.400,433.135,177.664,15.852,151.840
C06476=1100.385,179.650,433.113,177.668,15.853,151.840
C06477=1100.391,179.899,433.090,177.672,15.852,151.839
C06478=1100.396,180.147,433.067,177.675,15.851,151.838
C06479=1100.402,180.397,433.045,177.679,15.851,151.837
C06480=1100.408,180.646,433.023,177.682,15.851,151.836
C06481=1100.414,180.894,433.000,177.686,15.850,151.835
C06482=1100.419,181.143,432.977,177.689,15.849,151.835
C06483=1100.425,181.392,432.955,177.693,15.849,151.834
C06484=1100.430,181.641,432.932,177.697,15.849,151.833
C06485=1100.437,181.890,432.910,177.701,15.849,151.832
C06486=1100.442,182.139,432.887,177.704,15.848,151.831
C06487=1100.448,182.387,432.864,177.708,15.847,151.830
C06488=1100.454,182.637,432.842,177.711,15.847,151.829
C06489=1100.459,182.886,432.819,177.714,15.846,151.829
C06490=1100.466,183.134,432.796,177.718,15.846,151.828
C06491=1100.472,183.383,432.773,177.722,15.846,151.827
C06492=1100.477,183.632,432.750,177.726,15.845,151.826
C06493=1100.483,183.881,432.727,177.729,15.844,151.825
C06494=1100.488,184.131,432.705,177.733,15.844,151.824
C06495=1100.494,184.380,432.682,177.737,15.844,151.823
C06496=1100.500,184.628,432.659,177.740,15.843,151.823
C06497=1100.506,184.877,432.637,177.743,15.842,151.822
C06498=1100.512,185.126,432.614,177.747,15.842,151.821
C06499=1100.517,185.374,432.591,177.751,15.842,151.820
C06500=1100.523,185.623,432.568,177.754,15.841,151.819
C06501=1100.528,185.872,432.545,177.758,15.841,151.818
C06502=1100.534,186.121,432.522,177.761,15.841,151.818
C06503=1100.539,186.370,432.499,177.765,15.840,151.817
C06504=1100.545,186.619,432.476,177.769,15.840,151.816
C06505=1100.551,186.868,432.453,177.772,15.839,151.815
C06506=1100.557,187.117,432.430,177.776,15.839,151.814
C06507=1100.562,187.365,432.408,177.780,15.839,151.813
C06508=1100.567,187.614,432.384,177.783,15.838,151.812
C06509=1100.572,187.863,432.361,177.787,15.837,151.812
C06510=1100.578,188.112,432.338,177.790,15.837,151.811
C06511=1100.584,188.361,432.315,177.794,15.837,151.810
C06512=1100.590,188.610,432.292,177.798,15.837,151.809
C06513=1100.595,188.859,432.269,177.801,15.836,151.808
C06514=1100.600,189.108,432.246,177.805,15.835,151.807
C06515=1100.606,189.357,432.223,177.809,15.835,151.806
C06516=1100.612,189.606,432.200,177.812,15.835,151.806
C06517=1100.618,189.854,432.177,177.816,15.834,151.805
C06518=1100.623,190.104,432.153,177.819,15.834,151.804
C06519=1100.629,190.352,432.130,177.823,15.833,151.803
C06520=1100.634,190.601,432.107,177.827,15.833,151.802
C06521=1100.640,190.850,432.084,177.830,15.832,151.801
C06522=1100.645,191.099,432.060,177.834,15.832,151.800
C06523=1100.651,191.348,432.037,177.838,15.831,151.800
C06524=1100.657,191.596,432.014,177.841,15.831,151.799
C06525=1100.662,191.869,431.989,177.845,15.831,151.798
C06526=1100.668,192.142,431.963,177.849,15.830,151.797
C06527=1100.675,192.415,431.938,177.853,15.829,151.796
C06528=1100.681,192.688,431.912,177.857,15.829,151.795
C06529=1100.687,192.936,431.889,177.861,15.828,151.794
C06530=1100.692,193.185,431.865,177.864,15.827,151.793
C06531=1100.698,193.434,431.842,177.868,15.827,151.792
C06532=1100.704,193.683,431.819,177.872,15.827,151.791
C06533=1100.709,193.932,431.795,177.876,15.826,151.790
C06534=1100.715,194.181,431.772,177.880,15.826,151.790
C06535=1100.721,194.430,431.749,177.883,15.825,151.789
C06536=1100.726,194.678,431.725,177.887,15.825,151.788
C06537=1100.732,194.927,431.702,177.891,15.824,151.787
C06538=1100.737,195.176,431.679,177.894,15.824,151.786
C06539=1100.743,195.425,431.655,177.898,15.823,151.785
C06540=1100.749,195.674,431.631,177.901,15.823,151.784
C06541=1100.755,195.922,431.608,177.905,15.822,151.783
C06542=1100.760,196.172,431.584,177.909,15.822,151.783
C06543=1100.766,196.421,431.561,177.912,15.821,151.782
C06544=1100.772,196.669,431.538,177.916,15.821,151.781
C06545=1100.777,196.918,431.514,177.920,15.820,151.780
C06546=1100.783,197.166,431.490,177.924,15.820,151.779
C06547=1100.788,197.415,431.467,177.928,15.820,151.778
C06548=1100.794,197.665,431.443,177.931,15.818,151.777
C06549=1100.800,197.913,431.420,177.935,15.818,151.776
C06550=1100.805,198.162,431.396,177.939,15.817,151.775
C06551=1100.811,198.411,431.373,177.943,15.817,151.774
C06552=1100.817,198.659,431.349,177.946,15.816,151.774
C06553=1100.823,198.909,431.325,177.950,15.816,151.773
C06554=1100.829,199.157,431.301,177.953,15.816,151.772
C06555=1100.834,199.406,431.277,177.958,15.815,151.771
C06556=1100.840,199.655,431.254,177.961,15.814,151.770
C06557=1100.846,199.903,431.230,177.964,15.813,151.769
C06558=1100.851,200.153,431.207,177.968,15.813,151.768
C06559=1100.858,200.401,431.183,177.972,15.813,151.767
C06560=1100.863,200.650,431.159,177.976,15.812,151.766
C06561=1100.869,200.899,431.136,177.980,15.812,151.765
C06562=1100.874,201.147,431.111,177.983,15.811,151.765
C06563=1100.880,201.396,431.087,177.987,15.810,151.764
C06564=1100.885,201.646,431.064,177.991,15.810,151.763
C06565=1100.891,201.894,431.040,177.995,15.809,151.762
C06566=1100.898,202.142,431.017,177.998,15.808,151.761
C06567=1100.903,202.392,430.993,178.002,15.808,151.760
C06568=1100.909,202.640,430.969,178.006,15.807,151.759
C06569=1100.914,202.889,430.945,178.010,15.807,151.758
C06570=1100.920,203.139,430.921,178.014,15.807,151.757
C06571=1100.926,203.387,430.897,178.017,15.806,151.756
C06572=1100.931,203.636,430.873,178.021,15.805,151.755
C06573=1100.937,203.884,430.849,178.025,15.805,151.754
C06574=1100.943,204.133,430.825,178.029,15.804,151.753
C06575=1100.948,204.382,430.801,178.033,15.804,151.753
C06576=1100.954,204.631,430.777,178.036,15.803,151.752
C06577=1100.960,204.879,430.753,178.040,15.803,151.751
C06578=1100.965,205.128,430.729,178.044,15.802,151.750
C06579=1100.971,205.377,430.704,178.048,15.801,151.749
C06580=1100.977,205.626,430.681,178.052,15.801,151.748
C06581=1100.982,205.875,430.657,178.055,15.800,151.747
C06582=1100.988,206.124,430.632,178.059,15.799,151.746
C06583=1100.994,206.372,430.609,178.063,15.799,151.745
C06584=1100.999,206.621,430.585,178.067,15.799,151.744
C06585=1101.004,206.869,430.560,178.071,15.798,151.743
C06586=1101.011,207.118,430.536,178.075,15.798,151.742
C06587=1101.016,207.367,430.512,178.078,15.797,151.742
C06588=1101.022,207.616,430.488,178.081,15.796,151.741
C06589=1101.045,208.622,430.390,178.118,15.806,151.735
C06590=1101.053,208.990,430.354,178.124,15.806,151.734
C06591=1101.062,209.359,430.318,178.129,15.806,151.733
C06592=1101.070,209.728,430.281,178.134,15.807,151.732
C06593=1101.078,210.096,430.245,178.139,15.807,151.731
C06594=1101.085,210.345,430.221,178.144,15.808,151.730
C06595=1101.090,210.593,430.196,178.147,15.808,151.730
C06596=1101.095,210.842,430.172,178.151,15.809,151.729
C06597=1101.101,211.091,430.148,178.154,15.809,151.728
C06598=1101.106,211.340,430.123,178.158,15.809,151.728
C06599=1101.113,211.588,430.098,178.161,15.809,151.727
C06600=1101.118,211.837,430.074,178.164,15.810,151.726
C06601=1101.123,212.085,430.049,178.168,15.810,151.726
C06602=1101.129,212.335,430.025,178.171,15.810,151.725
C06603=1101.135,212.583,430.000,178.176,15.811,151.724
C06604=1101.141,212.832,429.975,178.179,15.811,151.723
C06605=1101.146,213.081,429.951,178.183,15.811,151.723
C06606=1101.152,213.329,429.926,178.186,15.811,151.722
C06607=1101.157,213.578,429.901,178.190,15.812,151.721
C06608=1101.163,213.827,429.877,178.193,15.812,151.721
C06609=1101.169,214.075,429.852,178.196,15.812,151.720
C06610=1101.173,214.324,429.827,178.200,15.812,151.719
C06611=1101.179,214.573,429.802,178.204,15.813,151.719
C06612=1101.185,214.821,429.777,178.208,15.813,151.718
C06613=1101.191,215.071,429.753,178.211,15.814,151.717
C06614=1101.196,215.319,429.728,178.215,15.814,151.717
C06615=1101.202,215.568,429.703,178.218,15.814,151.716
C06616=1101.208,215.816,429.679,178.222,15.814,151.715
C06617=1101.213,216.065,429.653,178.225,15.815,151.715
C06618=1101.218,216.314,429.629,178.229,15.816,151.714
C06619=1101.225,216.563,429.603,178.233,15.816,151.713
C06620=1101.230,216.811,429.579,178.236,15.816,151.713
C06621=1101.236,217.060,429.554,178.240,15.816,151.712
C06622=1101.241,217.308,429.530,178.243,15.817,151.711
C06623=1101.247,217.558,429.504,178.247,15.817,151.711
C06624=1101.252,217.806,429.479,178.250,15.817,151.710
C06625=1101.258,218.055,429.454,178.254,15.818,151.709
C06626=1101.264,218.304,429.429,178.258,15.818,151.709
C06627=1101.270,218.552,429.404,178.261,15.818,151.708
C06628=1101.275,218.802,429.379,178.265,15.819,151.707
C06629=1101.281,219.050,429.354,178.268,15.819,151.707
C06630=1101.287,219.299,429.330,178.272,15.819,151.706
C06631=1101.292,219.547,429.305,178.275,15.819,151.705
C06632=1101.298,219.796,429.279,178.279,15.820,151.705
C06633=1101.304,220.045,429.254,178.283,15.820,151.704
C06634=1101.309,220.293,429.229,178.286,15.821,151.703
C06635=1101.315,220.542,429.204,178.290,15.821,151.703
C06636=1101.320,220.791,429.179,178.293,15.821,151.702
C06637=1101.326,221.039,429.154,178.297,15.821,151.701
C06638=1101.332,221.288,429.128,178.301,15.822,151.700
C06639=1101.338,221.537,429.104,178.304,15.823,151.700
C06640=1101.343,221.785,429.078,178.308,15.823,151.699
C06641=1101.349,222.034,429.053,178.311,15.823,151.698
C06642=1101.358,222.407,429.015,178.317,15.824,151.697
C06643=1101.366,222.779,428.977,178.322,15.825,151.696
C06644=1101.374,223.151,428.939,178.327,15.825,151.695
C06645=1101.382,223.523,428.901,178.333,15.826,151.695
C06646=1101.388,223.773,428.877,178.336,15.826,151.694
C06647=1101.394,224.021,428.851,178.341,15.826,151.693
C06648=1101.399,224.269,428.826,178.344,15.827,151.693
C06649=1101.405,224.518,428.800,178.347,15.827,151.692
C06650=1101.411,224.767,428.775,178.351,15.827,151.691
C06651=1101.416,225.015,428.750,178.354,15.828,151.691
C06652=1101.422,225.264,428.724,178.358,15.829,151.690
C06653=1101.428,225.513,428.699,178.362,15.829,151.689
C06654=1101.433,225.762,428.673,178.366,15.829,151.688
C06655=1101.439,226.010,428.648,178.369,15.830,151.688
C06656=1101.444,226.259,428.622,178.372,15.830,151.687
C06657=1101.450,226.508,428.597,178.377,15.831,151.686
C06658=1101.455,226.756,428.571,178.380,15.831,151.686
C06659=1101.462,227.005,428.546,178.383,15.831,151.685
C06660=1101.467,227.254,428.520,178.387,15.832,151.685
C06661=1101.473,227.502,428.495,178.390,15.832,151.684
C06662=1101.478,227.751,428.469,178.394,15.833,151.683
C06663=1101.484,228.000,428.444,178.398,15.833,151.683
C06664=1101.490,228.249,428.418,178.402,15.833,151.682
C06665=1101.495,228.496,428.393,178.405,15.834,151.681
C06666=1101.501,228.745,428.367,178.408,15.834,151.681
C06667=1101.506,228.994,428.341,178.413,15.835,151.680
C06668=1101.512,229.243,428.316,178.416,15.835,151.679
C06669=1101.518,229.491,428.289,178.419,15.836,151.679
C06670=1101.524,229.739,428.264,178.423,15.836,151.678
C06671=1101.529,229.988,428.238,178.426,15.836,151.677
C06672=1101.536,230.237,428.213,178.430,15.837,151.677
C06673=1101.541,230.486,428.187,178.434,15.837,151.676
C06674=1101.546,230.735,428.161,178.438,15.837,151.675
C06675=1101.552,230.983,428.136,178.441,15.838,151.675
C06676=1101.558,231.231,428.109,178.445,15.839,151.674
C06677=1101.563,231.480,428.083,178.449,15.839,151.673
C06678=1101.569,231.729,428.057,178.452,15.840,151.673
C06679=1101.575,231.978,428.032,178.455,15.840,151.672
C06680=1101.580,232.226,428.006,178.460,15.841,151.671
C06681=1101.586,232.475,427.980,178.463,15.841,151.671
C06682=1101.591,232.724,427.954,178.466,15.841,151.670
C06683=1101.597,232.972,427.929,178.470,15.842,151.669
C06684=1101.603,233.221,427.903,178.474,15.843,151.669
C06685=1101.608,233.469,427.876,178.477,15.843,151.668
C06686=1101.613,233.718,427.850,178.481,15.843,151.667
C06687=1101.620,233.967,427.825,178.484,15.844,151.667
C06688=1101.625,234.215,427.798,178.488,15.844,151.666
C06689=1101.631,234.464,427.772,178.492,15.845,151.666
C06690=1101.636,234.713,427.747,178.495,15.845,151.665
C06691=1101.642,234.961,427.720,178.499,15.845,151.664
C06692=1101.647,235.210,427.694,178.503,15.847,151.664
C06693=1101.653,235.458,427.668,178.506,15.847,151.663
C06694=1101.661,235.822,427.630,178.512,15.848,151.662
C06695=1101.669,236.186,427.591,178.516,15.848,151.661
C06696=1101.678,236.550,427.554,178.522,15.849,151.660
C06697=1101.686,236.914,427.515,178.527,15.850,151.659
C06698=1101.691,237.163,427.489,178.531,15.850,151.659
C06699=1101.697,237.411,427.462,178.534,15.851,151.658
C06700=1101.703,237.660,427.437,178.538,15.851,151.657
C06701=1101.709,237.908,427.410,178.542,15.852,151.657
C06702=1101.715,238.157,427.384,178.545,15.852,151.656
C06703=1101.720,238.405,427.358,178.550,15.853,151.655
C06704=1101.726,238.654,427.332,178.553,15.854,151.655
C06705=1101.732,238.903,427.305,178.556,15.854,151.654
C06706=1101.737,239.151,427.279,178.559,15.854,151.654
C06707=1101.743,239.400,427.253,178.564,15.855,151.653
C06708=1101.749,239.648,427.226,178.567,15.855,151.652
C06709=1101.753,239.897,427.200,178.571,15.856,151.652
C06710=1101.759,240.145,427.174,178.575,15.857,151.651
C06711=1101.765,240.393,427.147,178.578,15.857,151.650
C06712=1101.770,240.642,427.121,178.582,15.858,151.650
C06713=1101.776,240.891,427.095,178.585,15.858,151.649
C06714=1101.782,241.139,427.068,178.589,15.859,151.648
C06715=1101.787,241.388,427.042,178.593,15.859,151.648
C06716=1101.793,241.636,427.015,178.596,15.860,151.647
C06717=1101.799,241.885,426.989,178.600,15.861,151.646
C06718=1101.805,242.133,426.962,178.604,15.861,151.646
C06719=1101.811,242.383,426.936,178.607,15.862,151.645
C06720=1101.817,242.631,426.909,178.610,15.862,151.644
C06721=1101.822,242.880,426.882,178.614,15.863,151.644
C06722=1101.828,243.128,426.856,178.618,15.863,151.643
C06723=1101.834,243.376,426.829,178.622,15.863,151.643
C06724=1101.839,243.626,426.803,178.625,15.865,151.642
C06725=1101.844,243.874,426.776,178.629,15.865,151.641
C06726=1101.850,244.122,426.749,178.632,15.865,151.641
C06727=1101.856,244.371,426.723,178.637,15.866,151.640
C06728=1101.862,244.619,426.696,178.640,15.867,151.640
C06729=1101.867,244.868,426.669,178.643,15.867,151.639
C06730=1101.872,245.117,426.643,178.647,15.868,151.638
C06731=1101.878,245.365,426.616,178.651,15.868,151.638
C06732=1101.884,245.613,426.590,178.654,15.869,151.637
C06733=1101.890,245.862,426.563,178.658,15.870,151.636
C06734=1101.895,246.110,426.536,178.662,15.871,151.636
C06735=1101.900,246.359,426.509,178.665,15.871,151.635
C06736=1101.906,246.607,426.482,178.669,15.872,151.635
C06737=1101.912,246.855,426.456,178.672,15.873,151.634
C06738=1101.917,247.104,426.428,178.676,15.873,151.633
C06739=1101.923,247.353,426.401,178.680,15.874,151.633
C06740=1101.929,247.602,426.375,178.683,15.874,151.632
C06741=1101.934,247.850,426.348,178.687,15.875,151.632
C06742=1101.940,248.099,426.321,178.691,15.876,151.631
C06743=1101.946,248.347,426.294,178.694,15.876,151.630
C06744=1101.951,248.596,426.267,178.697,15.877,151.630
C06745=1101.957,248.844,426.240,178.702,15.878,151.629
C06746=1101.964,249.201,426.202,178.706,15.878,151.628
C06747=1101.972,249.558,426.162,178.712,15.879,151.627
C06748=1101.981,249.915,426.123,178.717,15.880,151.626
C06749=1101.989,250.272,426.085,178.722,15.882,151.626
C06750=1101.994,250.521,426.058,178.726,15.882,151.625
C06751=1101.999,250.769,426.031,178.730,15.883,151.624
C06752=1102.005,251.018,426.004,178.733,15.883,151.624
C06753=1102.011,251.266,425.976,178.736,15.884,151.623
C06754=1102.017,251.515,425.949,178.740,15.885,151.623
C06755=1102.022,251.764,425.922,178.744,15.886,151.622
C06756=1102.028,252.012,425.895,178.747,15.886,151.621
C06757=1102.033,252.260,425.867,178.751,15.887,151.621
C06758=1102.039,252.508,425.841,178.754,15.888,151.620
C06759=1102.044,252.757,425.813,178.758,15.889,151.620
C06760=1102.051,253.005,425.786,178.762,15.889,151.619
C06761=1102.056,253.254,425.758,178.765,15.890,151.618
C06762=1102.061,253.503,425.732,178.769,15.891,151.618
C06763=1102.066,253.751,425.704,178.773,15.891,151.617
C06764=1102.072,253.999,425.677,178.776,15.892,151.617
C06765=1102.078,254.248,425.649,178.780,15.893,151.616
C06766=1102.084,254.496,425.622,178.783,15.893,151.615
C06767=1102.089,254.745,425.595,178.787,15.895,151.615
C06768=1102.095,254.993,425.568,178.791,15.895,151.614
C06769=1102.101,255.242,425.540,178.794,15.895,151.614
C06770=1102.106,255.490,425.513,178.798,15.897,151.613
C06771=1102.112,255.738,425.485,178.802,15.897,151.612
C06772=1102.117,255.987,425.458,178.806,15.898,151.612
C06773=1102.124,256.235,425.430,178.809,15.898,151.611
C06774=1102.129,256.484,425.403,178.812,15.899,151.611
C06775=1102.135,256.732,425.376,178.816,15.900,151.610
C06776=1102.141,256.981,425.348,178.820,15.901,151.609
C06777=1102.146,257.229,425.320,178.823,15.901,151.609
C06778=1102.152,257.478,425.294,178.827,15.902,151.608
C06779=1102.158,257.726,425.265,178.831,15.903,151.608
C06780=1102.163,257.975,425.238,178.835,15.904,151.607
C06781=1102.169,258.223,425.211,178.838,15.904,151.606
C06782=1102.175,258.471,425.182,178.841,15.905,151.606
C06783=1102.180,258.720,425.156,178.845,15.906,151.605
C06784=1102.186,258.968,425.128,178.849,15.906,151.605
C06785=1102.191,259.217,425.100,178.853,15.908,151.604
C06786=1102.197,259.465,425.073,178.856,15.908,151.604
C06787=1102.203,259.713,425.045,178.860,15.908,151.603
C06788=1102.208,259.962,425.017,178.864,15.910,151.602
C06789=1102.215,260.210,424.990,178.867,15.910,151.602
C06790=1102.220,260.458,424.962,178.871,15.911,151.601
C06791=1102.226,260.707,424.933,178.874,15.912,151.601
C06792=1102.232,260.955,424.907,178.878,15.913,151.600
C06793=1102.238,261.204,424.878,178.882,15.913,151.599
C06794=1102.243,261.452,424.851,178.885,15.914,151.599
C06795=1102.249,261.701,424.822,178.889,15.915,151.598
C06796=1102.255,261.949,424.796,178.893,15.915,151.598
C06797=1102.260,262.197,424.768,178.897,15.917,151.597
C06798=1102.269,262.551,424.728,178.902,15.918,151.596
C06799=1102.277,262.907,424.688,178.906,15.918,151.595
C06800=1102.285,263.260,424.649,178.912,15.919,151.595
C06801=1102.293,263.614,424.608,178.917,15.921,151.594
C06802=1102.299,263.862,424.581,178.921,15.922,151.593
C06803=1102.305,264.111,424.552,178.924,15.922,151.593
C06804=1102.310,264.360,424.525,178.928,15.923,151.592
C06805=1102.316,264.608,424.497,178.932,15.924,151.591
C06806=1102.321,264.856,424.469,178.935,15.925,151.591
C06807=1102.327,265.105,424.441,178.939,15.926,151.590
C06808=1102.333,265.353,424.413,178.942,15.926,151.590
C06809=1102.339,265.602,424.384,178.946,15.928,151.589
C06810=1102.344,265.850,424.356,178.950,15.928,151.589
C06811=1102.350,266.099,424.328,178.954,15.929,151.588
C06812=1102.355,266.347,424.300,178.957,15.930,151.588
C06813=1102.361,266.595,424.273,178.961,15.931,151.587
C06814=1102.367,266.843,424.244,178.964,15.932,151.586
C06815=1102.373,267.091,424.216,178.967,15.933,151.586
C06816=1102.378,267.340,424.188,178.972,15.933,151.585
C06817=1102.384,267.588,424.160,178.975,15.934,151.585
C06818=1102.390,267.836,424.131,178.979,15.935,151.584
C06819=1102.395,268.084,424.103,178.982,15.936,151.584
C06820=1102.401,268.333,424.074,178.986,15.937,151.583
C06821=1102.406,268.582,424.046,178.989,15.938,151.583
C06822=1102.412,268.830,424.018,178.993,15.939,151.582
C06823=1102.417,269.078,423.990,178.997,15.939,151.581
C06824=1102.423,269.327,423.962,179.001,15.941,151.581
C06825=1102.429,269.574,423.933,179.004,15.941,151.580
C06826=1102.435,269.823,423.905,179.008,15.943,151.580
C06827=1102.441,270.072,423.876,179.011,15.943,151.579
C06828=1102.446,270.320,423.848,179.015,15.945,151.579
C06829=1102.452,270.568,423.819,179.018,15.945,151.578
C06830=1102.458,270.816,423.791,179.022,15.947,151.578
C06831=1102.464,271.065,423.763,179.025,15.947,151.577
C06832=1102.468,271.313,423.734,179.030,15.948,151.577
C06833=1102.474,271.561,423.705,179.033,15.949,151.576
C06834=1102.480,271.810,423.677,179.036,15.949,151.575
C06835=1102.486,272.058,423.649,179.040,15.951,151.575
C06836=1102.492,272.306,423.620,179.043,15.951,151.574
C06837=1102.497,272.554,423.592,179.047,15.953,151.574
C06838=1102.503,272.804,423.563,179.051,15.953,151.573
C06839=1102.508,273.051,423.534,179.055,15.955,151.573
C06840=1102.514,273.300,423.506,179.058,15.955,151.572
C06841=1102.520,273.548,423.478,179.062,15.957,151.572
C06842=1102.526,273.796,423.449,179.065,15.957,151.571
C06843=1102.531,274.045,423.420,179.069,15.959,151.571
C06844=1102.537,274.292,423.392,179.073,15.960,151.570
C06845=1102.542,274.541,423.363,179.076,15.961,151.570
C06846=1102.549,274.789,423.334,179.080,15.962,151.569
C06847=1102.553,275.038,423.306,179.083,15.963,151.569
C06848=1102.560,275.286,423.277,179.087,15.964,151.568
C06849=1102.565,275.534,423.249,179.090,15.964,151.568
C06850=1102.573,275.892,423.207,179.096,15.966,151.567
C06851=1102.581,276.249,423.166,179.101,15.967,151.566
C06852=1102.590,276.605,423.124,179.106,15.969,151.565
C06853=1102.597,276.963,423.083,179.111,15.970,151.565
C06854=1102.603,277.211,423.054,179.115,15.971,151.564
C06855=1102.609,277.459,423.024,179.118,15.972,151.564
C06856=1102.614,277.707,422.996,179.122,15.973,151.563
C06857=1102.620,277.955,422.967,179.126,15.975,151.563
C06858=1102.626,278.204,422.938,179.129,15.975,151.562
C06859=1102.631,278.452,422.910,179.133,15.977,151.562
C06860=1102.637,278.700,422.880,179.136,15.977,151.561
C06861=1102.643,278.948,422.851,179.140,15.979,151.561
C06862=1102.648,279.196,422.823,179.143,15.980,151.560
C06863=1102.654,279.445,422.793,179.147,15.981,151.560
C06864=1102.660,279.693,422.764,179.151,15.982,151.559
C06865=1102.666,279.941,422.735,179.154,15.983,151.559
C06866=1102.671,280.189,422.707,179.158,15.984,151.558
C06867=1102.677,280.438,422.677,179.162,15.985,151.558
C06868=1102.683,280.686,422.648,179.166,15.986,151.557
C06869=1102.688,280.934,422.619,179.169,15.987,151.556
C06870=1102.694,281.182,422.590,179.172,15.989,151.556
C06871=1102.699,281.431,422.561,179.176,15.989,151.556
C06872=1102.705,281.679,422.532,179.180,15.991,151.555
C06873=1102.710,281.927,422.502,179.183,15.991,151.555
C06874=1102.717,282.175,422.473,179.187,15.993,151.554
C06875=1102.722,282.423,422.444,179.190,15.994,151.554
C06876=1102.728,282.672,422.414,179.194,15.995,151.553
C06877=1102.733,282.919,422.385,179.198,15.996,151.553
C06878=1102.739,283.168,422.356,179.201,15.997,151.552
C06879=1102.745,283.416,422.327,179.205,15.999,151.552
C06880=1102.750,283.665,422.298,179.208,16.000,151.551
C06881=1102.755,283.913,422.269,179.212,16.001,151.551
C06882=1102.761,284.161,422.240,179.216,16.002,151.550
C06883=1102.767,284.409,422.210,179.219,16.003,151.550
C06884=1102.772,284.658,422.180,179.223,16.005,151.549
C06885=1102.779,284.906,422.151,179.226,16.005,151.549
C06886=1102.784,285.154,422.122,179.229,16.007,151.548
C06887=1102.789,285.401,422.092,179.233,16.008,151.548
C06888=1102.796,285.650,422.063,179.237,16.009,151.547
C06889=1102.801,285.898,422.033,179.241,16.010,151.547
C06890=1102.807,286.146,422.003,179.243,16.011,151.547
C06891=1102.813,286.395,421.974,179.247,16.013,151.546
C06892=1102.818,286.642,421.945,179.251,16.013,151.546
C06893=1102.823,286.891,421.915,179.254,16.015,151.545
C06894=1102.829,287.139,421.886,179.258,16.016,151.545
C06895=1102.835,287.387,421.857,179.261,16.017,151.544
C06896=1102.841,287.635,421.826,179.265,16.018,151.544
C06897=1102.846,287.884,421.797,179.268,16.020,151.543
C06898=1102.852,288.132,421.767,179.272,16.021,151.543
C06899=1102.858,288.379,421.738,179.276,16.022,151.542
C06900=1102.863,288.628,421.709,179.279,16.023,151.542
C06901=1102.869,288.876,421.678,179.283,16.025,151.541
C06902=1102.878,289.242,421.635,179.288,16.026,151.541
C06903=1102.886,289.609,421.591,179.294,16.028,151.540
C06904=1102.895,289.975,421.547,179.299,16.030,151.539
C06905=1102.903,290.342,421.503,179.304,16.032,151.539
C06906=1102.908,290.590,421.473,179.308,16.033,151.538
C06907=1102.914,290.839,421.444,179.312,16.035,151.538
C06908=1102.920,291.086,421.414,179.315,16.036,151.537
C06909=1102.925,291.335,421.384,179.319,16.037,151.537
C06910=1102.931,291.583,421.354,179.322,16.039,151.537
C06911=1102.937,291.831,421.324,179.325,16.039,151.536
C06912=1102.943,292.079,421.295,179.329,16.041,151.536
C06913=1102.949,292.327,421.264,179.332,16.042,151.535
C06914=1102.953,292.575,421.235,179.336,16.044,151.535
C06915=1102.959,292.823,421.205,179.340,16.045,151.534
C06916=1102.965,293.071,421.175,179.343,16.046,151.534
C06917=1102.971,293.319,421.145,179.347,16.047,151.533
C06918=1102.976,293.567,421.115,179.350,16.049,151.533
C06919=1102.982,293.815,421.085,179.354,16.050,151.533
C06920=1102.987,294.064,421.055,179.357,16.051,151.532
C06921=1102.993,294.311,421.025,179.361,16.053,151.532
C06922=1102.999,294.560,420.995,179.364,16.054,151.531
C06923=1103.005,294.808,420.965,179.368,16.056,151.531
C06924=1103.010,295.055,420.935,179.372,16.057,151.531
C06925=1103.016,295.304,420.905,179.375,16.058,151.530
C06926=1103.022,295.552,420.875,179.379,16.059,151.530
C06927=1103.027,295.800,420.845,179.382,16.061,151.529
C06928=1103.033,296.048,420.815,179.385,16.062,151.529
C06929=1103.039,296.296,420.784,179.389,16.064,151.528
C06930=1103.044,296.545,420.754,179.393,16.065,151.528
C06931=1103.050,296.792,420.724,179.396,16.066,151.528
C06932=1103.055,297.040,420.693,179.400,16.068,151.527
C06933=1103.061,297.288,420.663,179.404,16.069,151.527
C06934=1103.067,297.536,420.633,179.407,16.071,151.526
C06935=1103.073,297.785,420.603,179.410,16.072,151.526
C06936=1103.079,298.033,420.572,179.414,16.073,151.526
C06937=1103.085,298.281,420.542,179.418,16.075,151.525
C06938=1103.089,298.529,420.512,179.421,16.076,151.525
C06939=1103.095,298.777,420.481,179.424,16.078,151.524
C06940=1103.101,299.025,420.451,179.428,16.079,151.524
C06941=1103.106,299.273,420.420,179.432,16.081,151.524
C06942=1103.112,299.521,420.390,179.435,16.082,151.523
C06943=1103.118,299.769,420.360,179.439,16.084,151.523
C06944=1103.123,300.017,420.330,179.442,16.086,151.523
C06945=1103.128,300.265,420.299,179.445,16.087,151.522
C06946=1103.134,300.513,420.268,179.449,16.088,151.522
C06947=1103.140,300.761,420.238,179.453,16.090,151.521
C06948=1103.145,301.009,420.207,179.456,16.092,151.521
C06949=1103.151,301.257,420.177,179.459,16.093,151.521
C06950=1103.157,301.505,420.146,179.463,16.094,151.520
C06951=1103.162,301.753,420.115,179.467,16.096,151.520
C06952=1103.168,302.001,420.085,179.470,16.098,151.520
C06953=1103.173,302.249,420.054,179.473,16.099,151.519
C06954=1103.182,302.629,420.008,179.479,16.101,151.519
C06955=1103.191,303.010,419.960,179.484,16.104,151.518
C06956=1103.199,303.391,419.914,179.490,16.107,151.518
C06957=1103.208,303.771,419.867,179.495,16.109,151.517
C06958=1103.213,304.019,419.836,179.498,16.110,151.517
C06959=1103.219,304.267,419.805,179.502,16.112,151.516
C06960=1103.224,304.515,419.774,179.506,16.114,151.516
C06961=1103.230,304.763,419.744,179.509,16.115,151.516
C06962=1103.236,305.011,419.712,179.512,16.116,151.515
C06963=1103.242,305.259,419.682,179.516,16.118,151.515
C06964=1103.247,305.506,419.651,179.520,16.120,151.515
C06965=1103.252,305.755,419.620,179.523,16.122,151.514
C06966=1103.258,306.002,419.590,179.526,16.123,151.514
C06967=1103.264,306.251,419.558,179.530,16.124,151.513
C06968=1103.270,306.498,419.528,179.534,16.126,151.513
C06969=1103.275,306.747,419.497,179.537,16.128,151.513
C06970=1103.281,306.994,419.466,179.541,16.130,151.512
C06971=1103.286,307.242,419.435,179.544,16.131,151.512
C06972=1103.293,307.490,419.404,179.547,16.133,151.512
C06973=1103.298,307.739,419.373,179.551,16.134,151.511
C06974=1103.304,307.986,419.343,179.555,16.136,151.511
C06975=1103.309,308.234,419.311,179.558,16.137,151.511
C06976=1103.315,308.482,419.280,179.561,16.139,151.510
C06977=1103.321,308.731,419.249,179.565,16.141,151.510
C06978=1103.327,308.978,419.218,179.569,16.142,151.510
C06979=1103.332,309.227,419.187,179.572,16.144,151.509
C06980=1103.338,309.474,419.155,179.575,16.146,151.509
C06981=1103.344,309.722,419.125,179.578,16.148,151.509
C06982=1103.349,309.971,419.094,179.582,16.149,151.509
C06983=1103.355,310.218,419.063,179.586,16.151,151.508
C06984=1103.360,310.466,419.032,179.589,16.153,151.508
C06985=1103.366,310.714,419.000,179.592,16.154,151.507
C06986=1103.372,310.962,418.969,179.596,16.156,151.507
C06987=1103.378,311.210,418.938,179.600,16.157,151.507
C06988=1103.384,311.458,418.907,179.603,16.159,151.506
C06989=1103.389,311.706,418.875,179.607,16.161,151.506
C06990=1103.395,311.954,418.844,179.610,16.163,151.506
C06991=1103.401,312.202,418.813,179.613,16.164,151.506
C06992=1103.406,312.450,418.782,179.617,16.166,151.505
C06993=1103.412,312.698,418.750,179.620,16.168,151.505
C06994=1103.418,312.945,418.719,179.624,16.170,151.505
C06995=1103.423,313.193,418.688,179.628,16.171,151.504
C06996=1103.430,313.441,418.657,179.630,16.173,151.504
C06997=1103.435,313.689,418.626,179.634,16.175,151.504
C06998=1103.441,313.938,418.594,179.638,16.176,151.503
C06999=1103.447,314.185,418.562,179.641,16.178,151.503
C07000=1103.453,314.434,418.531,179.645,16.180,151.503
C07001=1103.458,314.681,418.500,179.648,16.181,151.503
C07002=1103.464,314.929,418.467,179.651,16.183,151.502
C07003=1103.471,315.177,418.436,179.655,16.185,151.502
C07004=1103.476,315.425,418.405,179.659,16.187,151.502
C07005=1103.482,315.673,418.373,179.662,16.189,151.501
C07006=1103.489,316.056,418.325,179.667,16.192,151.501
C07007=1103.499,316.438,418.276,179.673,16.195,151.501
C07008=1103.507,316.822,418.227,179.678,16.198,151.500
C07009=1103.515,317.205,418.178,179.683,16.201,151.500
C07010=1103.521,317.453,418.146,179.686,16.203,151.499
C07011=1103.527,317.700,418.114,179.690,16.205,151.499
C07012=1103.532,317.948,418.083,179.693,16.206,151.499
C07013=1103.538,318.196,418.051,179.696,16.208,151.499
C07014=1103.543,318.444,418.020,179.699,16.210,151.499
C07015=1103.549,318.692,417.988,179.703,16.212,151.498
C07016=1103.554,318.940,417.956,179.706,16.214,151.498
C07017=1103.560,319.188,417.924,179.710,16.216,151.498
C07018=1103.566,319.436,417.892,179.713,16.218,151.498
C07019=1103.572,319.684,417.860,179.717,16.220,151.497
C07020=1103.577,319.931,417.829,179.720,16.222,151.497
C07021=1103.583,320.180,417.797,179.723,16.224,151.497
C07022=1103.589,320.427,417.765,179.726,16.226,151.497
C07023=1103.595,320.675,417.733,179.730,16.228,151.496
C07024=1103.600,320.923,417.701,179.733,16.230,151.496
C07025=1103.605,321.171,417.669,179.737,16.232,151.496
C07026=1103.611,321.419,417.637,179.740,16.234,151.496
C07027=1103.617,321.667,417.605,179.744,16.236,151.496
C07028=1103.622,321.915,417.573,179.747,16.238,151.495
C07029=1103.628,322.163,417.541,179.751,16.240,151.495
C07030=1103.633,322.410,417.510,179.754,16.242,151.495
C07031=1103.639,322.659,417.478,179.757,16.244,151.495
C07032=1103.646,322.906,417.445,179.761,16.246,151.495
C07033=1103.650,323.154,417.413,179.764,16.247,151.494
C07034=1103.656,323.402,417.381,179.767,16.250,151.494
C07035=1103.662,323.650,417.349,179.770,16.252,151.494
C07036=1103.668,323.898,417.317,179.774,16.254,151.494
C07037=1103.674,324.146,417.285,179.777,16.256,151.494
C07038=1103.679,324.393,417.252,179.781,16.258,151.493
C07039=1103.685,324.642,417.220,179.784,16.260,151.493
C07040=1103.690,324.889,417.188,179.787,16.262,151.493
C07041=1103.696,325.137,417.156,179.791,16.265,151.493
C07042=1103.702,325.385,417.123,179.794,16.267,151.493
C07043=1103.707,325.633,417.091,179.798,16.268,151.492
C07044=1103.713,325.881,417.059,179.801,16.271,151.492
C07045=1103.719,326.129,417.026,179.804,16.273,151.492
C07046=1103.725,326.376,416.995,179.808,16.275,151.492
C07047=1103.730,326.625,416.962,179.811,16.277,151.492
C07048=1103.736,326.872,416.929,179.814,16.279,151.491
C07049=1103.741,327.120,416.898,179.818,16.282,151.491
C07050=1103.747,327.368,416.866,179.821,16.284,151.491
C07051=1103.753,327.616,416.832,179.825,16.286,151.491
C07052=1103.759,327.864,416.800,179.828,16.288,151.491
C07053=1103.765,328.111,416.768,179.831,16.290,151.490
C07054=1103.771,328.359,416.736,179.835,16.292,151.490
C07055=1103.776,328.608,416.703,179.838,16.294,151.490
C07056=1103.782,328.855,416.671,179.841,16.296,151.490
C07057=1103.788,329.103,416.639,179.845,16.299,151.490
C07058=1103.796,329.478,416.589,179.850,16.302,151.490
C07059=1103.805,329.854,416.539,179.855,16.305,151.489
C07060=1103.814,330.230,416.490,179.860,16.309,151.489
C07061=1103.822,330.607,416.441,179.865,16.312,151.489
C07062=1103.828,330.853,416.408,179.868,16.314,151.489
C07063=1103.834,331.102,416.376,179.872,16.316,151.488
C07064=1103.840,331.350,416.343,179.875,16.318,151.488
C07065=1103.846,331.597,416.310,179.878,16.321,151.488
C07066=1103.851,331.846,416.277,179.882,16.323,151.488
C07067=1103.858,332.093,416.245,179.885,16.325,151.488
C07068=1103.863,332.340,416.212,179.888,16.327,151.488
C07069=1103.869,332.589,416.180,179.891,16.330,151.488
C07070=1103.874,332.837,416.146,179.895,16.332,151.487
C07071=1103.880,333.084,416.114,179.898,16.334,151.487
C07072=1103.886,333.333,416.081,179.901,16.337,151.487
C07073=1103.891,333.580,416.049,179.904,16.339,151.487
C07074=1103.897,333.828,416.015,179.907,16.341,151.487
C07075=1103.902,334.075,415.982,179.911,16.344,151.487
C07076=1103.908,334.324,415.950,179.914,16.346,151.487
C07077=1103.914,334.572,415.917,179.918,16.349,151.487
C07078=1103.920,334.818,415.884,179.921,16.351,151.487
C07079=1103.925,335.066,415.851,179.924,16.354,151.487
C07080=1103.931,335.314,415.818,179.928,16.356,151.486
C07081=1103.937,335.562,415.786,179.931,16.358,151.486
C07082=1103.942,335.810,415.752,179.934,16.361,151.486
C07083=1103.948,336.058,415.719,179.937,16.363,151.486
C07084=1103.954,336.305,415.686,179.940,16.366,151.486
C07085=1103.959,336.553,415.653,179.944,16.368,151.486
C07086=1103.965,336.801,415.620,179.947,16.370,151.486
C07087=1103.971,337.049,415.587,179.950,16.373,151.486
C07088=1103.976,337.296,415.554,179.954,16.376,151.486
C07089=1103.982,337.544,415.520,179.957,16.378,151.486
C07090=1103.988,337.792,415.488,179.960,16.381,151.486
C07091=1103.994,338.040,415.454,179.964,16.383,151.485
C07092=1103.999,338.288,415.421,179.967,16.385,151.485
C07093=1104.005,338.536,415.388,179.970,16.388,151.485
C07094=1104.011,338.783,415.355,179.973,16.390,151.485
C07095=1104.016,339.030,415.322,179.976,16.393,151.485
C07096=1104.022,339.278,415.289,179.980,16.395,151.485
C07097=1104.027,339.526,415.255,179.983,16.398,151.485
C07098=1104.033,339.774,415.222,179.986,16.401,151.485
C07099=1104.038,340.022,415.189,179.989,16.403,151.485
C07100=1104.045,340.269,415.155,179.993,16.406,151.485
C07101=1104.051,340.517,415.122,179.996,16.408,151.485
C07102=1104.056,340.765,415.088,179.999,16.411,151.485
C07103=1104.062,341.013,415.055,-179.997,16.414,151.485
C07104=1104.067,341.261,415.022,-179.994,16.417,151.485
C07105=1104.073,341.509,414.988,-179.991,16.419,151.485
C07106=1104.079,341.756,414.954,-179.988,16.421,151.485
C07107=1104.084,342.004,414.921,-179.985,16.424,151.485
C07108=1104.090,342.252,414.888,-179.982,16.427,151.485
C07109=1104.095,342.499,414.855,-179.978,16.430,151.485
C07110=1104.104,342.868,414.804,-179.973,16.434,151.485
C07111=1104.113,343.239,414.754,-179.969,16.437,151.485
C07112=1104.121,343.608,414.704,-179.964,16.441,151.485
C07113=1104.130,343.978,414.655,-179.959,16.446,151.485
C07114=1104.135,344.226,414.621,-179.956,16.448,151.485
C07115=1104.141,344.473,414.587,-179.953,16.451,151.485
C07116=1104.147,344.721,414.554,-179.949,16.453,151.485
C07117=1104.153,344.968,414.520,-179.946,16.456,151.485
C07118=1104.158,345.216,414.486,-179.943,16.459,151.485
C07119=1104.164,345.463,414.452,-179.940,16.462,151.485
C07120=1104.170,345.711,414.419,-179.937,16.464,151.485
C07121=1104.175,345.959,414.386,-179.934,16.467,151.485
C07122=1104.180,346.207,414.351,-179.930,16.471,151.485
C07123=1104.186,346.455,414.318,-179.927,16.473,151.485
C07124=1104.192,346.702,414.284,-179.924,16.476,151.485
C07125=1104.198,346.949,414.250,-179.921,16.478,151.485
C07126=1104.203,347.197,414.216,-179.918,16.481,151.485
C07127=1104.210,347.445,414.182,-179.914,16.485,151.485
C07128=1104.215,347.693,414.149,-179.911,16.487,151.485
C07129=1104.221,347.940,414.115,-179.908,16.490,151.485
C07130=1104.226,348.188,414.081,-179.905,16.493,151.485
C07131=1104.232,348.436,414.047,-179.902,16.496,151.485
C07132=1104.238,348.683,414.012,-179.899,16.499,151.485
C07133=1104.243,348.931,413.979,-179.896,16.501,151.485
C07134=1104.249,349.178,413.945,-179.892,16.505,151.485
C07135=1104.254,349.426,413.910,-179.889,16.507,151.485
C07136=1104.260,349.674,413.877,-179.886,16.510,151.485
C07137=1104.266,349.921,413.843,-179.883,16.513,151.485
C07138=1104.272,350.169,413.809,-179.879,16.516,151.485
C07139=1104.277,350.417,413.774,-179.877,16.519,151.486
C07140=1104.283,350.664,413.741,-179.874,16.522,151.486
C07141=1104.289,350.912,413.707,-179.870,16.526,151.486
C07142=1104.294,351.159,413.673,-179.867,16.528,151.486
C07143=1104.300,351.407,413.638,-179.864,16.531,151.486
C07144=1104.305,351.655,413.605,-179.861,16.534,151.486
C07145=1104.312,351.903,413.570,-179.858,16.537,151.486
C07146=1104.317,352.150,413.536,-179.855,16.540,151.486
C07147=1104.323,352.397,413.501,-179.852,16.543,151.486
C07148=1104.328,352.645,413.467,-179.848,16.547,151.487
C07149=1104.334,352.892,413.433,-179.845,16.549,151.487
C07150=1104.340,353.140,413.398,-179.843,16.552,151.487
C07151=1104.346,353.388,413.364,-179.839,16.555,151.487
C07152=1104.352,353.635,413.330,-179.836,16.558,151.487
C07153=1104.357,353.882,413.296,-179.833,16.561,151.487
C07154=1104.363,354.130,413.261,-179.830,16.565,151.487
C07155=1104.368,354.377,413.227,-179.827,16.568,151.487
C07156=1104.374,354.625,413.192,-179.824,16.571,151.487
C07157=1104.379,354.873,413.158,-179.820,16.574,151.488
C07158=1104.385,355.120,413.124,-179.818,16.577,151.488
C07159=1104.391,355.367,413.090,-179.814,16.581,151.488
C07160=1104.397,355.616,413.055,-179.811,16.584,151.488
C07161=1104.403,355.863,413.021,-179.809,16.587,151.488
C07162=1104.411,356.235,412.969,-179.804,16.592,151.488
C07163=1104.419,356.607,412.918,-179.799,16.596,151.489
C07164=1104.428,356.978,412.865,-179.795,16.601,151.489
C07165=1104.436,357.351,412.814,-179.790,16.606,151.489
C07166=1104.442,357.598,412.779,-179.787,16.609,151.489
C07167=1104.448,357.846,412.744,-179.784,16.612,151.489
C07168=1104.453,358.093,412.709,-179.781,16.616,151.490
C07169=1104.459,358.341,412.674,-179.778,16.619,151.490
C07170=1104.465,358.589,412.640,-179.775,16.623,151.490
C07171=1104.470,358.836,412.605,-179.772,16.626,151.490
C07172=1104.476,359.083,412.571,-179.769,16.629,151.490
C07173=1104.481,359.331,412.536,-179.766,16.633,151.491
C07174=1104.488,359.579,412.502,-179.763,16.636,151.491
C07175=1104.493,359.826,412.466,-179.759,16.639,151.491
C07176=1104.498,360.073,412.432,-179.757,16.642,151.491
C07177=1104.505,360.321,412.397,-179.753,16.646,151.491
C07178=1104.510,360.568,412.362,-179.751,16.649,151.492
C07179=1104.516,360.816,412.328,-179.748,16.652,151.492
C07180=1104.522,361.063,412.292,-179.745,16.656,151.492
C07181=1104.527,361.311,412.257,-179.742,16.659,151.492
C07182=1104.532,361.558,412.223,-179.738,16.663,151.492
C07183=1104.539,361.806,412.188,-179.736,16.666,151.493
C07184=1104.544,362.053,412.153,-179.732,16.670,151.493
C07185=1104.550,362.300,412.118,-179.730,16.673,151.493
C07186=1104.556,362.548,412.083,-179.726,16.677,151.493
C07187=1104.562,362.795,412.048,-179.724,16.680,151.494
C07188=1104.567,363.043,412.013,-179.720,16.684,151.494
C07189=1104.573,363.291,411.977,-179.718,16.687,151.494
C07190=1104.579,363.538,411.943,-179.715,16.691,151.494
C07191=1104.585,363.785,411.908,-179.712,16.695,151.495
C07192=1104.590,364.032,411.872,-179.709,16.698,151.495
C07193=1104.595,364.280,411.838,-179.706,16.702,151.495
C07194=1104.601,364.528,411.802,-179.703,16.705,151.495
C07195=1104.607,364.775,411.768,-179.700,16.709,151.496
C07196=1104.613,365.023,411.732,-179.698,16.712,151.496
C07197=1104.619,365.270,411.697,-179.694,16.716,151.496
C07198=1104.624,365.517,411.662,-179.692,16.719,151.497
C07199=1104.630,365.765,411.626,-179.688,16.723,151.497
C07200=1104.635,366.012,411.591,-179.686,16.726,151.497
C07201=1104.642,366.259,411.556,-179.682,16.730,151.497
C07202=1104.647,366.507,411.521,-179.679,16.734,151.498
C07203=1104.653,366.755,411.485,-179.677,16.738,151.498
C07204=1104.659,367.002,411.450,-179.673,16.742,151.498
C07205=1104.664,367.248,411.415,-179.671,16.745,151.499
C07206=1104.670,367.497,411.380,-179.668,16.749,151.499
C07207=1104.675,367.744,411.344,-179.665,16.752,151.499
C07208=1104.681,367.991,411.309,-179.662,16.756,151.500
C07209=1104.687,368.238,411.273,-179.660,16.760,151.500
C07210=1104.693,368.486,411.238,-179.656,16.764,151.500
C07211=1104.698,368.733,411.202,-179.653,16.768,151.501
C07212=1104.703,368.981,411.168,-179.651,16.771,151.501
C07213=1104.709,369.228,411.132,-179.648,16.776,151.502
C07214=1104.718,369.615,411.076,-179.643,16.781,151.502
C07215=1104.727,370.002,411.020,-179.639,16.787,151.503
C07216=1104.736,370.388,410.965,-179.635,16.793,151.503
C07217=1104.745,370.775,410.909,-179.630,16.799,151.504
C07218=1104.750,371.022,410.873,-179.627,16.803,151.504
C07219=1104.756,371.270,410.837,-179.624,16.807,151.505
C07220=1104.762,371.517,410.802,-179.622,16.811,151.505
C07221=1104.768,371.764,410.766,-179.619,16.815,151.505
C07222=1104.773,372.011,410.731,-179.616,16.819,151.506
C07223=1104.779,372.259,410.695,-179.613,16.823,151.506
C07224=1104.785,372.507,410.660,-179.610,16.827,151.507
C07225=1104.790,372.754,410.624,-179.607,16.830,151.507
C07226=1104.796,373.002,410.588,-179.605,16.835,151.507
C07227=1104.801,373.248,410.552,-179.601,16.839,151.508
C07228=1104.808,373.496,410.516,-179.599,16.843,151.508
C07229=1104.813,373.743,410.481,-179.596,16.847,151.509
C07230=1104.819,373.990,410.445,-179.593,16.851,151.509
C07231=1104.825,374.238,410.409,-179.590,16.855,151.509
C07232=1104.831,374.484,410.373,-179.587,16.859,151.510
C07233=1104.836,374.732,410.337,-179.585,16.863,151.510
C07234=1104.841,374.979,410.301,-179.582,16.867,151.511
C07235=1104.848,375.226,410.265,-179.579,16.871,151.511
C07236=1104.852,375.474,410.229,-179.576,16.876,151.512
C07237=1104.859,375.721,410.193,-179.574,16.879,151.512
C07238=1104.865,375.969,410.158,-179.571,16.884,151.513
C07239=1104.870,376.216,410.121,-179.568,16.888,151.513
C07240=1104.876,376.463,410.085,-179.566,16.892,151.514
C07241=1104.881,376.710,410.049,-179.563,16.896,151.514
C07242=1104.887,376.958,410.013,-179.560,16.900,151.515
C07243=1104.893,377.205,409.977,-179.558,16.904,151.515
C07244=1104.898,377.452,409.941,-179.555,16.909,151.516
C07245=1104.904,377.700,409.905,-179.552,16.913,151.516
C07246=1104.909,377.946,409.869,-179.549,16.918,151.517
C07247=1104.915,378.194,409.833,-179.547,16.922,151.517
C07248=1104.921,378.441,409.796,-179.544,16.926,151.518
C07249=1104.926,378.688,409.760,-179.541,16.930,151.518
C07250=1104.932,378.935,409.723,-179.538,16.935,151.519
C07251=1104.938,379.183,409.688,-179.536,16.939,151.519
C07252=1104.944,379.429,409.652,-179.533,16.943,151.520
C07253=1104.949,379.677,409.615,-179.530,16.948,151.520
C07254=1104.955,379.925,409.579,-179.527,16.952,151.521
C07255=1104.960,380.171,409.542,-179.525,16.956,151.521
C07256=1104.966,380.419,409.506,-179.522,16.961,151.522
C07257=1104.972,380.666,409.469,-179.519,16.965,151.522
C07258=1104.978,380.913,409.433,-179.516,16.970,151.523
C07259=1104.983,381.161,409.397,-179.515,16.974,151.524
C07260=1104.989,381.408,409.361,-179.512,16.978,151.524
C07261=1104.996,381.655,409.324,-179.509,16.983,151.525
C07262=1105.000,381.902,409.288,-179.506,16.988,151.525
C07263=1105.007,382.149,409.252,-179.503,16.992,151.526
